  PROC Part96()
    MoveL Offs(pOrigin,43.0,16.5,15.0),vTravel,z5,tPen\WObj:=wPaper;
    MoveL Offs(pOrigin,43.0,16.5,0.0),vApproach,fine,tPen\WObj:=wPaper;
    MoveL Offs(pOrigin,42.8,16.3,0.0),vDraw,z1,tPen\WObj:=wPaper;
    MoveL Offs(pOrigin,42.6,16.5,0.0),vDraw,z1,tPen\WObj:=wPaper;
    MoveL Offs(pOrigin,42.6,18.2,0.0),vDraw,z1,tPen\WObj:=wPaper;
    MoveL Offs(pOrigin,42.8,18.4,0.0),vDraw,z1,tPen\WObj:=wPaper;
    MoveL Offs(pOrigin,43.0,18.2,0.0),vDraw,z1,tPen\WObj:=wPaper;
    MoveL Offs(pOrigin,43.0,17.7,0.0),vDraw,z1,tPen\WObj:=wPaper;
    MoveL Offs(pOrigin,43.2,17.5,0.0),vDraw,z1,tPen\WObj:=wPaper;
    MoveL Offs(pOrigin,43.0,17.3,0.0),vDraw,z1,tPen\WObj:=wPaper;
    MoveL Offs(pOrigin,43.0,16.5,0.0),vDraw,fine,tPen\WObj:=wPaper;
    MoveL Offs(pOrigin,43.0,16.5,15.0),vApproach,z5,tPen\WObj:=wPaper;
    MoveL Offs(pOrigin,43.2,18.4,15.0),vTravel,z5,tPen\WObj:=wPaper;
    MoveL Offs(pOrigin,43.2,18.4,0.0),vApproach,fine,tPen\WObj:=wPaper;
    MoveL Offs(pOrigin,43.0,18.6,0.0),vDraw,z1,tPen\WObj:=wPaper;
    MoveL Offs(pOrigin,43.8,19.2,0.0),vDraw,z1,tPen\WObj:=wPaper;
    MoveL Offs(pOrigin,44.0,19.2,0.0),vDraw,z1,tPen\WObj:=wPaper;
    MoveL Offs(pOrigin,44.2,19.0,0.0),vDraw,z1,tPen\WObj:=wPaper;
    MoveL Offs(pOrigin,44.2,18.8,0.0),vDraw,z1,tPen\WObj:=wPaper;
    MoveL Offs(pOrigin,44.0,18.6,0.0),vDraw,z1,tPen\WObj:=wPaper;
    MoveL Offs(pOrigin,43.6,18.6,0.0),vDraw,z1,tPen\WObj:=wPaper;
    MoveL Offs(pOrigin,43.4,18.4,0.0),vDraw,z1,tPen\WObj:=wPaper;
    MoveL Offs(pOrigin,43.2,18.4,0.0),vDraw,fine,tPen\WObj:=wPaper;
    MoveL Offs(pOrigin,43.2,18.4,15.0),vApproach,z5,tPen\WObj:=wPaper;
    MoveL Offs(pOrigin,46.0,19.0,15.0),vTravel,z5,tPen\WObj:=wPaper;
    MoveL Offs(pOrigin,46.0,19.0,0.0),vApproach,fine,tPen\WObj:=wPaper;
    MoveL Offs(pOrigin,46.2,19.2,0.0),vDraw,z1,tPen\WObj:=wPaper;
    MoveL Offs(pOrigin,46.8,19.2,0.0),vDraw,z1,tPen\WObj:=wPaper;
    MoveL Offs(pOrigin,47.0,19.4,0.0),vDraw,z1,tPen\WObj:=wPaper;
    MoveL Offs(pOrigin,47.6,19.4,0.0),vDraw,z1,tPen\WObj:=wPaper;
    MoveL Offs(pOrigin,47.7,19.5,0.0),vDraw,z1,tPen\WObj:=wPaper;
    MoveL Offs(pOrigin,47.9,19.4,0.0),vDraw,z1,tPen\WObj:=wPaper;
    MoveL Offs(pOrigin,47.9,19.0,0.0),vDraw,z1,tPen\WObj:=wPaper;
    MoveL Offs(pOrigin,47.7,18.8,0.0),vDraw,z1,tPen\WObj:=wPaper;
    MoveL Offs(pOrigin,46.2,18.8,0.0),vDraw,z1,tPen\WObj:=wPaper;
    MoveL Offs(pOrigin,46.0,19.0,0.0),vDraw,fine,tPen\WObj:=wPaper;
    MoveL Offs(pOrigin,46.0,19.0,15.0),vApproach,z5,tPen\WObj:=wPaper;
    MoveL Offs(pOrigin,48.1,19.5,15.0),vTravel,z5,tPen\WObj:=wPaper;
    MoveL Offs(pOrigin,48.1,19.5,0.0),vApproach,fine,tPen\WObj:=wPaper;
    MoveL Offs(pOrigin,48.3,19.7,0.0),vDraw,z1,tPen\WObj:=wPaper;
    MoveL Offs(pOrigin,48.9,19.7,0.0),vDraw,z1,tPen\WObj:=wPaper;
    MoveL Offs(pOrigin,49.1,19.9,0.0),vDraw,z1,tPen\WObj:=wPaper;
    MoveL Offs(pOrigin,49.3,19.9,0.0),vDraw,z1,tPen\WObj:=wPaper;
    MoveL Offs(pOrigin,49.4,19.7,0.0),vDraw,z1,tPen\WObj:=wPaper;
    MoveL Offs(pOrigin,49.4,19.5,0.0),vDraw,z1,tPen\WObj:=wPaper;
    MoveL Offs(pOrigin,49.3,19.4,0.0),vDraw,z1,tPen\WObj:=wPaper;
    MoveL Offs(pOrigin,48.3,19.4,0.0),vDraw,z1,tPen\WObj:=wPaper;
    MoveL Offs(pOrigin,48.1,19.5,0.0),vDraw,fine,tPen\WObj:=wPaper;
    MoveL Offs(pOrigin,48.1,19.5,15.0),vApproach,z5,tPen\WObj:=wPaper;
    MoveL Offs(pOrigin,46.6,26.3,15.0),vTravel,z5,tPen\WObj:=wPaper;
    MoveL Offs(pOrigin,46.6,26.3,0.0),vApproach,fine,tPen\WObj:=wPaper;
    MoveL Offs(pOrigin,46.4,26.5,0.0),vDraw,z1,tPen\WObj:=wPaper;
    MoveL Offs(pOrigin,46.4,27.1,0.0),vDraw,z1,tPen\WObj:=wPaper;
    MoveL Offs(pOrigin,46.2,27.3,0.0),vDraw,z1,tPen\WObj:=wPaper;
    MoveL Offs(pOrigin,46.2,29.9,0.0),vDraw,z1,tPen\WObj:=wPaper;
    MoveL Offs(pOrigin,45.9,30.5,0.0),vDraw,z1,tPen\WObj:=wPaper;
    MoveL Offs(pOrigin,46.0,30.7,0.0),vDraw,z1,tPen\WObj:=wPaper;
    MoveL Offs(pOrigin,46.6,30.7,0.0),vDraw,z1,tPen\WObj:=wPaper;
    MoveL Offs(pOrigin,46.8,30.5,0.0),vDraw,z1,tPen\WObj:=wPaper;
    MoveL Offs(pOrigin,46.8,30.3,0.0),vDraw,z1,tPen\WObj:=wPaper;
    MoveL Offs(pOrigin,46.6,30.1,0.0),vDraw,z1,tPen\WObj:=wPaper;
    MoveL Offs(pOrigin,46.6,28.6,0.0),vDraw,z1,tPen\WObj:=wPaper;
    MoveL Offs(pOrigin,46.8,28.6,0.0),vDraw,z1,tPen\WObj:=wPaper;
    MoveL Offs(pOrigin,47.0,28.4,0.0),vDraw,z1,tPen\WObj:=wPaper;
    MoveL Offs(pOrigin,47.0,27.9,0.0),vDraw,z1,tPen\WObj:=wPaper;
    MoveL Offs(pOrigin,46.8,27.7,0.0),vDraw,z1,tPen\WObj:=wPaper;
    MoveL Offs(pOrigin,46.8,26.5,0.0),vDraw,z1,tPen\WObj:=wPaper;
    MoveL Offs(pOrigin,46.6,26.3,0.0),vDraw,fine,tPen\WObj:=wPaper;
    MoveL Offs(pOrigin,46.6,26.3,15.0),vApproach,z5,tPen\WObj:=wPaper;
    MoveL Offs(pOrigin,47.2,29.0,15.0),vTravel,z5,tPen\WObj:=wPaper;
    MoveL Offs(pOrigin,47.2,29.0,0.0),vApproach,fine,tPen\WObj:=wPaper;
    MoveL Offs(pOrigin,47.0,29.2,0.0),vDraw,z1,tPen\WObj:=wPaper;
    MoveL Offs(pOrigin,47.0,29.7,0.0),vDraw,z1,tPen\WObj:=wPaper;
    MoveL Offs(pOrigin,47.4,30.3,0.0),vDraw,z1,tPen\WObj:=wPaper;
    MoveL Offs(pOrigin,47.6,30.1,0.0),vDraw,z1,tPen\WObj:=wPaper;
    MoveL Offs(pOrigin,47.6,29.7,0.0),vDraw,z1,tPen\WObj:=wPaper;
    MoveL Offs(pOrigin,47.4,29.6,0.0),vDraw,z1,tPen\WObj:=wPaper;
    MoveL Offs(pOrigin,47.4,29.2,0.0),vDraw,z1,tPen\WObj:=wPaper;
    MoveL Offs(pOrigin,47.2,29.0,0.0),vDraw,fine,tPen\WObj:=wPaper;
    MoveL Offs(pOrigin,47.2,29.0,15.0),vApproach,z5,tPen\WObj:=wPaper;
    MoveL Offs(pOrigin,46.4,31.6,15.0),vTravel,z5,tPen\WObj:=wPaper;
    MoveL Offs(pOrigin,46.4,31.6,0.0),vApproach,fine,tPen\WObj:=wPaper;
    MoveL Offs(pOrigin,46.2,31.8,0.0),vDraw,z1,tPen\WObj:=wPaper;
    MoveL Offs(pOrigin,46.2,32.2,0.0),vDraw,z1,tPen\WObj:=wPaper;
    MoveL Offs(pOrigin,46.0,32.4,0.0),vDraw,z1,tPen\WObj:=wPaper;
    MoveL Offs(pOrigin,46.0,33.0,0.0),vDraw,z1,tPen\WObj:=wPaper;
    MoveL Offs(pOrigin,45.9,33.1,0.0),vDraw,z1,tPen\WObj:=wPaper;
    MoveL Offs(pOrigin,45.9,33.9,0.0),vDraw,z1,tPen\WObj:=wPaper;
    MoveL Offs(pOrigin,45.7,34.1,0.0),vDraw,z1,tPen\WObj:=wPaper;
    MoveL Offs(pOrigin,45.7,35.0,0.0),vDraw,z1,tPen\WObj:=wPaper;
    MoveL Offs(pOrigin,45.5,35.2,0.0),vDraw,z1,tPen\WObj:=wPaper;
    MoveL Offs(pOrigin,45.5,37.3,0.0),vDraw,z1,tPen\WObj:=wPaper;
    MoveL Offs(pOrigin,45.7,37.5,0.0),vDraw,z1,tPen\WObj:=wPaper;
    MoveL Offs(pOrigin,45.7,38.1,0.0),vDraw,z1,tPen\WObj:=wPaper;
    MoveL Offs(pOrigin,45.9,38.2,0.0),vDraw,z1,tPen\WObj:=wPaper;
    MoveL Offs(pOrigin,45.9,38.8,0.0),vDraw,z1,tPen\WObj:=wPaper;
    MoveL Offs(pOrigin,46.0,39.0,0.0),vDraw,z1,tPen\WObj:=wPaper;
    MoveL Offs(pOrigin,46.0,39.2,0.0),vDraw,z1,tPen\WObj:=wPaper;
    MoveL Offs(pOrigin,46.2,39.4,0.0),vDraw,z1,tPen\WObj:=wPaper;
    MoveL Offs(pOrigin,46.8,40.7,0.0),vDraw,z1,tPen\WObj:=wPaper;
    MoveL Offs(pOrigin,47.4,41.5,0.0),vDraw,z1,tPen\WObj:=wPaper;
    MoveL Offs(pOrigin,47.6,41.3,0.0),vDraw,z1,tPen\WObj:=wPaper;
    MoveL Offs(pOrigin,47.6,40.7,0.0),vDraw,z1,tPen\WObj:=wPaper;
    MoveL Offs(pOrigin,48.3,40.7,0.0),vDraw,z1,tPen\WObj:=wPaper;
    MoveL Offs(pOrigin,48.5,40.5,0.0),vDraw,z1,tPen\WObj:=wPaper;
    MoveL Offs(pOrigin,47.6,39.6,0.0),vDraw,z1,tPen\WObj:=wPaper;
    MoveL Offs(pOrigin,47.6,39.4,0.0),vDraw,z1,tPen\WObj:=wPaper;
    MoveL Offs(pOrigin,46.6,38.2,0.0),vDraw,z1,tPen\WObj:=wPaper;
    MoveL Offs(pOrigin,46.6,38.1,0.0),vDraw,z1,tPen\WObj:=wPaper;
    MoveL Offs(pOrigin,46.4,37.9,0.0),vDraw,z1,tPen\WObj:=wPaper;
    MoveL Offs(pOrigin,46.4,37.5,0.0),vDraw,z1,tPen\WObj:=wPaper;
    MoveL Offs(pOrigin,45.9,36.5,0.0),vDraw,z1,tPen\WObj:=wPaper;
    MoveL Offs(pOrigin,45.9,35.4,0.0),vDraw,z1,tPen\WObj:=wPaper;
    MoveL Offs(pOrigin,46.6,35.4,0.0),vDraw,z1,tPen\WObj:=wPaper;
    MoveL Offs(pOrigin,46.6,35.6,0.0),vDraw,z1,tPen\WObj:=wPaper;
    MoveL Offs(pOrigin,46.8,35.8,0.0),vDraw,z1,tPen\WObj:=wPaper;
    MoveL Offs(pOrigin,47.4,37.1,0.0),vDraw,z1,tPen\WObj:=wPaper;
    MoveL Offs(pOrigin,47.7,37.5,0.0),vDraw,z1,tPen\WObj:=wPaper;
    MoveL Offs(pOrigin,47.7,37.7,0.0),vDraw,z1,tPen\WObj:=wPaper;
    MoveL Offs(pOrigin,48.1,38.1,0.0),vDraw,z1,tPen\WObj:=wPaper;
  ENDPROC

  PROC Part97()
    MoveL Offs(pOrigin,48.1,38.2,0.0),vDraw,z1,tPen\WObj:=wPaper;
    MoveL Offs(pOrigin,51.1,41.3,0.0),vDraw,z1,tPen\WObj:=wPaper;
    MoveL Offs(pOrigin,51.3,41.3,0.0),vDraw,z1,tPen\WObj:=wPaper;
    MoveL Offs(pOrigin,52.3,42.2,0.0),vDraw,z1,tPen\WObj:=wPaper;
    MoveL Offs(pOrigin,52.5,42.2,0.0),vDraw,z1,tPen\WObj:=wPaper;
    MoveL Offs(pOrigin,53.0,42.8,0.0),vDraw,z1,tPen\WObj:=wPaper;
    MoveL Offs(pOrigin,53.2,42.8,0.0),vDraw,z1,tPen\WObj:=wPaper;
    MoveL Offs(pOrigin,53.4,42.6,0.0),vDraw,z1,tPen\WObj:=wPaper;
    MoveL Offs(pOrigin,52.5,41.5,0.0),vDraw,z1,tPen\WObj:=wPaper;
    MoveL Offs(pOrigin,52.5,41.3,0.0),vDraw,z1,tPen\WObj:=wPaper;
    MoveL Offs(pOrigin,51.7,40.3,0.0),vDraw,z1,tPen\WObj:=wPaper;
    MoveL Offs(pOrigin,51.5,39.8,0.0),vDraw,z1,tPen\WObj:=wPaper;
    MoveL Offs(pOrigin,51.1,39.4,0.0),vDraw,z1,tPen\WObj:=wPaper;
    MoveL Offs(pOrigin,51.1,39.2,0.0),vDraw,z1,tPen\WObj:=wPaper;
    MoveL Offs(pOrigin,50.2,37.5,0.0),vDraw,z1,tPen\WObj:=wPaper;
    MoveL Offs(pOrigin,50.2,37.1,0.0),vDraw,z1,tPen\WObj:=wPaper;
    MoveL Offs(pOrigin,49.8,36.7,0.0),vDraw,z1,tPen\WObj:=wPaper;
    MoveL Offs(pOrigin,49.6,36.7,0.0),vDraw,z1,tPen\WObj:=wPaper;
    MoveL Offs(pOrigin,49.4,36.9,0.0),vDraw,z1,tPen\WObj:=wPaper;
    MoveL Offs(pOrigin,49.1,36.9,0.0),vDraw,z1,tPen\WObj:=wPaper;
    MoveL Offs(pOrigin,49.1,36.7,0.0),vDraw,z1,tPen\WObj:=wPaper;
    MoveL Offs(pOrigin,48.5,36.0,0.0),vDraw,z1,tPen\WObj:=wPaper;
    MoveL Offs(pOrigin,48.5,35.8,0.0),vDraw,z1,tPen\WObj:=wPaper;
    MoveL Offs(pOrigin,48.3,35.6,0.0),vDraw,z1,tPen\WObj:=wPaper;
    MoveL Offs(pOrigin,48.3,35.4,0.0),vDraw,z1,tPen\WObj:=wPaper;
    MoveL Offs(pOrigin,48.1,35.2,0.0),vDraw,z1,tPen\WObj:=wPaper;
    MoveL Offs(pOrigin,48.1,35.0,0.0),vDraw,z1,tPen\WObj:=wPaper;
    MoveL Offs(pOrigin,47.9,34.8,0.0),vDraw,z1,tPen\WObj:=wPaper;
    MoveL Offs(pOrigin,47.9,34.7,0.0),vDraw,z1,tPen\WObj:=wPaper;
    MoveL Offs(pOrigin,46.8,32.6,0.0),vDraw,z1,tPen\WObj:=wPaper;
    MoveL Offs(pOrigin,46.8,32.2,0.0),vDraw,z1,tPen\WObj:=wPaper;
    MoveL Offs(pOrigin,46.4,31.6,0.0),vDraw,fine,tPen\WObj:=wPaper;
    MoveL Offs(pOrigin,46.4,31.6,15.0),vApproach,z5,tPen\WObj:=wPaper;
    MoveL Offs(pOrigin,45.1,33.5,15.0),vTravel,z5,tPen\WObj:=wPaper;
    MoveL Offs(pOrigin,45.1,33.5,0.0),vApproach,fine,tPen\WObj:=wPaper;
    MoveL Offs(pOrigin,44.9,33.7,0.0),vDraw,z1,tPen\WObj:=wPaper;
    MoveL Offs(pOrigin,44.9,34.7,0.0),vDraw,z1,tPen\WObj:=wPaper;
    MoveL Offs(pOrigin,45.1,34.8,0.0),vDraw,z1,tPen\WObj:=wPaper;
    MoveL Offs(pOrigin,45.3,34.7,0.0),vDraw,z1,tPen\WObj:=wPaper;
    MoveL Offs(pOrigin,45.3,33.7,0.0),vDraw,z1,tPen\WObj:=wPaper;
    MoveL Offs(pOrigin,45.1,33.5,0.0),vDraw,fine,tPen\WObj:=wPaper;
    MoveL Offs(pOrigin,45.1,33.5,15.0),vApproach,z5,tPen\WObj:=wPaper;
    MoveL Offs(pOrigin,44.9,34.7,15.0),vTravel,z5,tPen\WObj:=wPaper;
    MoveL Offs(pOrigin,44.9,34.7,0.0),vApproach,fine,tPen\WObj:=wPaper;
    MoveL Offs(pOrigin,44.7,34.8,0.0),vDraw,z1,tPen\WObj:=wPaper;
    MoveL Offs(pOrigin,44.7,37.5,0.0),vDraw,z1,tPen\WObj:=wPaper;
    MoveL Offs(pOrigin,44.9,37.7,0.0),vDraw,z1,tPen\WObj:=wPaper;
    MoveL Offs(pOrigin,45.1,37.5,0.0),vDraw,z1,tPen\WObj:=wPaper;
    MoveL Offs(pOrigin,45.1,34.8,0.0),vDraw,z1,tPen\WObj:=wPaper;
    MoveL Offs(pOrigin,44.9,34.7,0.0),vDraw,fine,tPen\WObj:=wPaper;
    MoveL Offs(pOrigin,44.9,34.7,15.0),vApproach,z5,tPen\WObj:=wPaper;
    MoveL Offs(pOrigin,57.4,15.6,15.0),vTravel,z5,tPen\WObj:=wPaper;
    MoveL Offs(pOrigin,57.4,15.6,0.0),vApproach,fine,tPen\WObj:=wPaper;
    MoveL Offs(pOrigin,58.3,15.6,0.0),vDraw,z1,tPen\WObj:=wPaper;
    MoveL Offs(pOrigin,58.5,15.4,0.0),vDraw,z1,tPen\WObj:=wPaper;
    MoveL Offs(pOrigin,58.3,15.2,0.0),vDraw,z1,tPen\WObj:=wPaper;
    MoveL Offs(pOrigin,57.4,15.2,0.0),vDraw,z1,tPen\WObj:=wPaper;
    MoveL Offs(pOrigin,57.2,15.4,0.0),vDraw,z1,tPen\WObj:=wPaper;
    MoveL Offs(pOrigin,57.4,15.6,0.0),vDraw,fine,tPen\WObj:=wPaper;
    MoveL Offs(pOrigin,57.4,15.6,15.0),vApproach,z5,tPen\WObj:=wPaper;
    MoveL Offs(pOrigin,57.4,14.8,15.0),vTravel,z5,tPen\WObj:=wPaper;
    MoveL Offs(pOrigin,57.4,14.8,0.0),vApproach,fine,tPen\WObj:=wPaper;
    MoveL Offs(pOrigin,58.7,14.8,0.0),vDraw,z1,tPen\WObj:=wPaper;
    MoveL Offs(pOrigin,58.9,14.6,0.0),vDraw,z1,tPen\WObj:=wPaper;
    MoveL Offs(pOrigin,58.7,14.4,0.0),vDraw,z1,tPen\WObj:=wPaper;
    MoveL Offs(pOrigin,57.4,14.4,0.0),vDraw,z1,tPen\WObj:=wPaper;
    MoveL Offs(pOrigin,57.2,14.6,0.0),vDraw,z1,tPen\WObj:=wPaper;
    MoveL Offs(pOrigin,57.4,14.8,0.0),vDraw,fine,tPen\WObj:=wPaper;
    MoveL Offs(pOrigin,57.4,14.8,15.0),vApproach,z5,tPen\WObj:=wPaper;
    MoveL Offs(pOrigin,59.1,14.4,15.0),vTravel,z5,tPen\WObj:=wPaper;
    MoveL Offs(pOrigin,59.1,14.4,0.0),vApproach,fine,tPen\WObj:=wPaper;
    MoveL Offs(pOrigin,59.3,14.6,0.0),vDraw,z1,tPen\WObj:=wPaper;
    MoveL Offs(pOrigin,60.6,14.6,0.0),vDraw,z1,tPen\WObj:=wPaper;
    MoveL Offs(pOrigin,60.8,14.4,0.0),vDraw,z1,tPen\WObj:=wPaper;
    MoveL Offs(pOrigin,60.6,14.3,0.0),vDraw,z1,tPen\WObj:=wPaper;
    MoveL Offs(pOrigin,59.3,14.3,0.0),vDraw,z1,tPen\WObj:=wPaper;
    MoveL Offs(pOrigin,59.1,14.4,0.0),vDraw,fine,tPen\WObj:=wPaper;
    MoveL Offs(pOrigin,59.1,14.4,15.0),vApproach,z5,tPen\WObj:=wPaper;
    MoveL Offs(pOrigin,59.3,15.0,15.0),vTravel,z5,tPen\WObj:=wPaper;
    MoveL Offs(pOrigin,59.3,15.0,0.0),vApproach,fine,tPen\WObj:=wPaper;
    MoveL Offs(pOrigin,59.1,15.2,0.0),vDraw,z1,tPen\WObj:=wPaper;
    MoveL Offs(pOrigin,59.3,15.4,0.0),vDraw,z1,tPen\WObj:=wPaper;
    MoveL Offs(pOrigin,60.2,15.4,0.0),vDraw,z1,tPen\WObj:=wPaper;
    MoveL Offs(pOrigin,60.4,15.2,0.0),vDraw,z1,tPen\WObj:=wPaper;
    MoveL Offs(pOrigin,60.2,15.0,0.0),vDraw,z1,tPen\WObj:=wPaper;
    MoveL Offs(pOrigin,59.3,15.0,0.0),vDraw,fine,tPen\WObj:=wPaper;
    MoveL Offs(pOrigin,59.3,15.0,15.0),vApproach,z5,tPen\WObj:=wPaper;
    MoveL Offs(pOrigin,61.0,15.0,15.0),vTravel,z5,tPen\WObj:=wPaper;
    MoveL Offs(pOrigin,61.0,15.0,0.0),vApproach,fine,tPen\WObj:=wPaper;
    MoveL Offs(pOrigin,61.2,15.2,0.0),vDraw,z1,tPen\WObj:=wPaper;
    MoveL Offs(pOrigin,61.9,15.2,0.0),vDraw,z1,tPen\WObj:=wPaper;
    MoveL Offs(pOrigin,62.1,15.0,0.0),vDraw,z1,tPen\WObj:=wPaper;
    MoveL Offs(pOrigin,61.9,14.8,0.0),vDraw,z1,tPen\WObj:=wPaper;
    MoveL Offs(pOrigin,61.2,14.8,0.0),vDraw,z1,tPen\WObj:=wPaper;
    MoveL Offs(pOrigin,61.0,15.0,0.0),vDraw,fine,tPen\WObj:=wPaper;
    MoveL Offs(pOrigin,61.0,15.0,15.0),vApproach,z5,tPen\WObj:=wPaper;
    MoveL Offs(pOrigin,61.2,14.4,15.0),vTravel,z5,tPen\WObj:=wPaper;
    MoveL Offs(pOrigin,61.2,14.4,0.0),vApproach,fine,tPen\WObj:=wPaper;
    MoveL Offs(pOrigin,62.5,14.4,0.0),vDraw,z1,tPen\WObj:=wPaper;
    MoveL Offs(pOrigin,62.7,14.3,0.0),vDraw,z1,tPen\WObj:=wPaper;
    MoveL Offs(pOrigin,62.5,14.1,0.0),vDraw,z1,tPen\WObj:=wPaper;
    MoveL Offs(pOrigin,61.2,14.1,0.0),vDraw,z1,tPen\WObj:=wPaper;
    MoveL Offs(pOrigin,61.0,14.3,0.0),vDraw,z1,tPen\WObj:=wPaper;
    MoveL Offs(pOrigin,61.2,14.4,0.0),vDraw,fine,tPen\WObj:=wPaper;
    MoveL Offs(pOrigin,61.2,14.4,15.0),vApproach,z5,tPen\WObj:=wPaper;
    MoveL Offs(pOrigin,62.9,14.1,15.0),vTravel,z5,tPen\WObj:=wPaper;
    MoveL Offs(pOrigin,62.9,14.1,0.0),vApproach,fine,tPen\WObj:=wPaper;
    MoveL Offs(pOrigin,63.0,14.3,0.0),vDraw,z1,tPen\WObj:=wPaper;
    MoveL Offs(pOrigin,64.4,14.3,0.0),vDraw,z1,tPen\WObj:=wPaper;
    MoveL Offs(pOrigin,64.6,14.1,0.0),vDraw,z1,tPen\WObj:=wPaper;
    MoveL Offs(pOrigin,64.4,13.9,0.0),vDraw,z1,tPen\WObj:=wPaper;
    MoveL Offs(pOrigin,63.0,13.9,0.0),vDraw,z1,tPen\WObj:=wPaper;
    MoveL Offs(pOrigin,62.9,14.1,0.0),vDraw,fine,tPen\WObj:=wPaper;
    MoveL Offs(pOrigin,62.9,14.1,15.0),vApproach,z5,tPen\WObj:=wPaper;
    MoveL Offs(pOrigin,63.0,14.6,15.0),vTravel,z5,tPen\WObj:=wPaper;
    MoveL Offs(pOrigin,63.0,14.6,0.0),vApproach,fine,tPen\WObj:=wPaper;
    MoveL Offs(pOrigin,62.9,14.8,0.0),vDraw,z1,tPen\WObj:=wPaper;
    MoveL Offs(pOrigin,63.0,15.0,0.0),vDraw,z1,tPen\WObj:=wPaper;
    MoveL Offs(pOrigin,63.8,15.0,0.0),vDraw,z1,tPen\WObj:=wPaper;
    MoveL Offs(pOrigin,64.0,14.8,0.0),vDraw,z1,tPen\WObj:=wPaper;
  ENDPROC

  PROC Part98()
    MoveL Offs(pOrigin,63.8,14.6,0.0),vDraw,z1,tPen\WObj:=wPaper;
    MoveL Offs(pOrigin,63.0,14.6,0.0),vDraw,fine,tPen\WObj:=wPaper;
    MoveL Offs(pOrigin,63.0,14.6,15.0),vApproach,z5,tPen\WObj:=wPaper;
    MoveL Offs(pOrigin,64.7,14.6,15.0),vTravel,z5,tPen\WObj:=wPaper;
    MoveL Offs(pOrigin,64.7,14.6,0.0),vApproach,fine,tPen\WObj:=wPaper;
    MoveL Offs(pOrigin,64.9,14.8,0.0),vDraw,z1,tPen\WObj:=wPaper;
    MoveL Offs(pOrigin,65.7,14.8,0.0),vDraw,z1,tPen\WObj:=wPaper;
    MoveL Offs(pOrigin,65.9,14.6,0.0),vDraw,z1,tPen\WObj:=wPaper;
    MoveL Offs(pOrigin,65.7,14.4,0.0),vDraw,z1,tPen\WObj:=wPaper;
    MoveL Offs(pOrigin,64.9,14.4,0.0),vDraw,z1,tPen\WObj:=wPaper;
    MoveL Offs(pOrigin,64.7,14.6,0.0),vDraw,fine,tPen\WObj:=wPaper;
    MoveL Offs(pOrigin,64.7,14.6,15.0),vApproach,z5,tPen\WObj:=wPaper;
    MoveL Offs(pOrigin,64.9,14.1,15.0),vTravel,z5,tPen\WObj:=wPaper;
    MoveL Offs(pOrigin,64.9,14.1,0.0),vApproach,fine,tPen\WObj:=wPaper;
    MoveL Offs(pOrigin,66.1,14.1,0.0),vDraw,z1,tPen\WObj:=wPaper;
    MoveL Offs(pOrigin,66.3,13.9,0.0),vDraw,z1,tPen\WObj:=wPaper;
    MoveL Offs(pOrigin,66.1,13.7,0.0),vDraw,z1,tPen\WObj:=wPaper;
    MoveL Offs(pOrigin,64.9,13.7,0.0),vDraw,z1,tPen\WObj:=wPaper;
    MoveL Offs(pOrigin,64.7,13.9,0.0),vDraw,z1,tPen\WObj:=wPaper;
    MoveL Offs(pOrigin,64.9,14.1,0.0),vDraw,fine,tPen\WObj:=wPaper;
    MoveL Offs(pOrigin,64.9,14.1,15.0),vApproach,z5,tPen\WObj:=wPaper;
    MoveL Offs(pOrigin,66.4,13.7,15.0),vTravel,z5,tPen\WObj:=wPaper;
    MoveL Offs(pOrigin,66.4,13.7,0.0),vApproach,fine,tPen\WObj:=wPaper;
    MoveL Offs(pOrigin,66.6,13.9,0.0),vDraw,z1,tPen\WObj:=wPaper;
    MoveL Offs(pOrigin,68.0,13.9,0.0),vDraw,z1,tPen\WObj:=wPaper;
    MoveL Offs(pOrigin,68.1,13.7,0.0),vDraw,z1,tPen\WObj:=wPaper;
    MoveL Offs(pOrigin,68.0,13.5,0.0),vDraw,z1,tPen\WObj:=wPaper;
    MoveL Offs(pOrigin,66.6,13.5,0.0),vDraw,z1,tPen\WObj:=wPaper;
    MoveL Offs(pOrigin,66.4,13.7,0.0),vDraw,fine,tPen\WObj:=wPaper;
    MoveL Offs(pOrigin,66.4,13.7,15.0),vApproach,z5,tPen\WObj:=wPaper;
    MoveL Offs(pOrigin,66.6,14.3,15.0),vTravel,z5,tPen\WObj:=wPaper;
    MoveL Offs(pOrigin,66.6,14.3,0.0),vApproach,fine,tPen\WObj:=wPaper;
    MoveL Offs(pOrigin,66.4,14.4,0.0),vDraw,z1,tPen\WObj:=wPaper;
    MoveL Offs(pOrigin,66.6,14.6,0.0),vDraw,z1,tPen\WObj:=wPaper;
    MoveL Offs(pOrigin,67.6,14.6,0.0),vDraw,z1,tPen\WObj:=wPaper;
    MoveL Offs(pOrigin,67.8,14.4,0.0),vDraw,z1,tPen\WObj:=wPaper;
    MoveL Offs(pOrigin,67.6,14.3,0.0),vDraw,z1,tPen\WObj:=wPaper;
    MoveL Offs(pOrigin,66.6,14.3,0.0),vDraw,fine,tPen\WObj:=wPaper;
    MoveL Offs(pOrigin,66.6,14.3,15.0),vApproach,z5,tPen\WObj:=wPaper;
    MoveL Offs(pOrigin,66.4,15.6,15.0),vTravel,z5,tPen\WObj:=wPaper;
    MoveL Offs(pOrigin,66.4,15.6,0.0),vApproach,fine,tPen\WObj:=wPaper;
    MoveL Offs(pOrigin,66.3,15.8,0.0),vDraw,z1,tPen\WObj:=wPaper;
    MoveL Offs(pOrigin,66.4,16.0,0.0),vDraw,z1,tPen\WObj:=wPaper;
    MoveL Offs(pOrigin,67.2,16.0,0.0),vDraw,z1,tPen\WObj:=wPaper;
    MoveL Offs(pOrigin,67.4,15.8,0.0),vDraw,z1,tPen\WObj:=wPaper;
    MoveL Offs(pOrigin,67.2,15.6,0.0),vDraw,z1,tPen\WObj:=wPaper;
    MoveL Offs(pOrigin,66.4,15.6,0.0),vDraw,fine,tPen\WObj:=wPaper;
    MoveL Offs(pOrigin,66.4,15.6,15.0),vApproach,z5,tPen\WObj:=wPaper;
    MoveL Offs(pOrigin,65.5,16.0,15.0),vTravel,z5,tPen\WObj:=wPaper;
    MoveL Offs(pOrigin,65.5,16.0,0.0),vApproach,fine,tPen\WObj:=wPaper;
    MoveL Offs(pOrigin,65.3,15.8,0.0),vDraw,z1,tPen\WObj:=wPaper;
    MoveL Offs(pOrigin,64.6,15.8,0.0),vDraw,z1,tPen\WObj:=wPaper;
    MoveL Offs(pOrigin,64.4,16.0,0.0),vDraw,z1,tPen\WObj:=wPaper;
    MoveL Offs(pOrigin,64.6,16.1,0.0),vDraw,z1,tPen\WObj:=wPaper;
    MoveL Offs(pOrigin,65.3,16.1,0.0),vDraw,z1,tPen\WObj:=wPaper;
    MoveL Offs(pOrigin,65.5,16.0,0.0),vDraw,fine,tPen\WObj:=wPaper;
    MoveL Offs(pOrigin,65.5,16.0,15.0),vApproach,z5,tPen\WObj:=wPaper;
    MoveL Offs(pOrigin,68.1,15.6,15.0),vTravel,z5,tPen\WObj:=wPaper;
    MoveL Offs(pOrigin,68.1,15.6,0.0),vApproach,fine,tPen\WObj:=wPaper;
    MoveL Offs(pOrigin,68.3,15.8,0.0),vDraw,z1,tPen\WObj:=wPaper;
    MoveL Offs(pOrigin,69.1,15.8,0.0),vDraw,z1,tPen\WObj:=wPaper;
    MoveL Offs(pOrigin,69.3,15.6,0.0),vDraw,z1,tPen\WObj:=wPaper;
    MoveL Offs(pOrigin,69.1,15.4,0.0),vDraw,z1,tPen\WObj:=wPaper;
    MoveL Offs(pOrigin,68.3,15.4,0.0),vDraw,z1,tPen\WObj:=wPaper;
    MoveL Offs(pOrigin,68.1,15.6,0.0),vDraw,fine,tPen\WObj:=wPaper;
    MoveL Offs(pOrigin,68.1,15.6,15.0),vApproach,z5,tPen\WObj:=wPaper;
    MoveL Offs(pOrigin,68.5,14.4,15.0),vTravel,z5,tPen\WObj:=wPaper;
    MoveL Offs(pOrigin,68.5,14.4,0.0),vApproach,fine,tPen\WObj:=wPaper;
    MoveL Offs(pOrigin,69.3,14.4,0.0),vDraw,z1,tPen\WObj:=wPaper;
    MoveL Offs(pOrigin,69.5,14.3,0.0),vDraw,z1,tPen\WObj:=wPaper;
    MoveL Offs(pOrigin,69.3,14.1,0.0),vDraw,z1,tPen\WObj:=wPaper;
    MoveL Offs(pOrigin,68.5,14.1,0.0),vDraw,z1,tPen\WObj:=wPaper;
    MoveL Offs(pOrigin,68.3,14.3,0.0),vDraw,z1,tPen\WObj:=wPaper;
    MoveL Offs(pOrigin,68.5,14.4,0.0),vDraw,fine,tPen\WObj:=wPaper;
    MoveL Offs(pOrigin,68.5,14.4,15.0),vApproach,z5,tPen\WObj:=wPaper;
    MoveL Offs(pOrigin,68.3,13.7,15.0),vTravel,z5,tPen\WObj:=wPaper;
    MoveL Offs(pOrigin,68.3,13.7,0.0),vApproach,fine,tPen\WObj:=wPaper;
    MoveL Offs(pOrigin,69.7,13.7,0.0),vDraw,z1,tPen\WObj:=wPaper;
    MoveL Offs(pOrigin,69.8,13.5,0.0),vDraw,z1,tPen\WObj:=wPaper;
    MoveL Offs(pOrigin,69.7,13.3,0.0),vDraw,z1,tPen\WObj:=wPaper;
    MoveL Offs(pOrigin,68.3,13.3,0.0),vDraw,z1,tPen\WObj:=wPaper;
    MoveL Offs(pOrigin,68.1,13.5,0.0),vDraw,z1,tPen\WObj:=wPaper;
    MoveL Offs(pOrigin,68.3,13.7,0.0),vDraw,fine,tPen\WObj:=wPaper;
    MoveL Offs(pOrigin,68.3,13.7,15.0),vApproach,z5,tPen\WObj:=wPaper;
    MoveL Offs(pOrigin,70.0,13.3,15.0),vTravel,z5,tPen\WObj:=wPaper;
    MoveL Offs(pOrigin,70.0,13.3,0.0),vApproach,fine,tPen\WObj:=wPaper;
    MoveL Offs(pOrigin,70.2,13.5,0.0),vDraw,z1,tPen\WObj:=wPaper;
    MoveL Offs(pOrigin,71.5,13.5,0.0),vDraw,z1,tPen\WObj:=wPaper;
    MoveL Offs(pOrigin,71.7,13.3,0.0),vDraw,z1,tPen\WObj:=wPaper;
    MoveL Offs(pOrigin,71.5,13.1,0.0),vDraw,z1,tPen\WObj:=wPaper;
    MoveL Offs(pOrigin,70.2,13.1,0.0),vDraw,z1,tPen\WObj:=wPaper;
    MoveL Offs(pOrigin,70.0,13.3,0.0),vDraw,fine,tPen\WObj:=wPaper;
    MoveL Offs(pOrigin,70.0,13.3,15.0),vApproach,z5,tPen\WObj:=wPaper;
    MoveL Offs(pOrigin,70.2,13.9,15.0),vTravel,z5,tPen\WObj:=wPaper;
    MoveL Offs(pOrigin,70.2,13.9,0.0),vApproach,fine,tPen\WObj:=wPaper;
    MoveL Offs(pOrigin,70.0,14.1,0.0),vDraw,z1,tPen\WObj:=wPaper;
    MoveL Offs(pOrigin,70.2,14.3,0.0),vDraw,z1,tPen\WObj:=wPaper;
    MoveL Offs(pOrigin,71.2,14.3,0.0),vDraw,z1,tPen\WObj:=wPaper;
    MoveL Offs(pOrigin,71.4,14.1,0.0),vDraw,z1,tPen\WObj:=wPaper;
    MoveL Offs(pOrigin,71.2,13.9,0.0),vDraw,z1,tPen\WObj:=wPaper;
    MoveL Offs(pOrigin,70.2,13.9,0.0),vDraw,fine,tPen\WObj:=wPaper;
    MoveL Offs(pOrigin,70.2,13.9,15.0),vApproach,z5,tPen\WObj:=wPaper;
    MoveL Offs(pOrigin,70.2,15.2,15.0),vTravel,z5,tPen\WObj:=wPaper;
    MoveL Offs(pOrigin,70.2,15.2,0.0),vApproach,fine,tPen\WObj:=wPaper;
    MoveL Offs(pOrigin,70.0,15.4,0.0),vDraw,z1,tPen\WObj:=wPaper;
    MoveL Offs(pOrigin,70.2,15.6,0.0),vDraw,z1,tPen\WObj:=wPaper;
    MoveL Offs(pOrigin,71.2,15.6,0.0),vDraw,z1,tPen\WObj:=wPaper;
    MoveL Offs(pOrigin,71.4,15.4,0.0),vDraw,z1,tPen\WObj:=wPaper;
    MoveL Offs(pOrigin,71.2,15.2,0.0),vDraw,z1,tPen\WObj:=wPaper;
    MoveL Offs(pOrigin,70.2,15.2,0.0),vDraw,fine,tPen\WObj:=wPaper;
    MoveL Offs(pOrigin,70.2,15.2,15.0),vApproach,z5,tPen\WObj:=wPaper;
    MoveL Offs(pOrigin,71.9,15.2,15.0),vTravel,z5,tPen\WObj:=wPaper;
    MoveL Offs(pOrigin,71.9,15.2,0.0),vApproach,fine,tPen\WObj:=wPaper;
    MoveL Offs(pOrigin,72.1,15.4,0.0),vDraw,z1,tPen\WObj:=wPaper;
    MoveL Offs(pOrigin,73.1,15.4,0.0),vDraw,z1,tPen\WObj:=wPaper;
    MoveL Offs(pOrigin,73.2,15.2,0.0),vDraw,z1,tPen\WObj:=wPaper;
    MoveL Offs(pOrigin,73.1,15.0,0.0),vDraw,z1,tPen\WObj:=wPaper;
    MoveL Offs(pOrigin,72.1,15.0,0.0),vDraw,z1,tPen\WObj:=wPaper;
    MoveL Offs(pOrigin,71.9,15.2,0.0),vDraw,fine,tPen\WObj:=wPaper;
    MoveL Offs(pOrigin,71.9,15.2,15.0),vApproach,z5,tPen\WObj:=wPaper;
  ENDPROC

  PROC Part99()
    MoveL Offs(pOrigin,72.1,14.1,15.0),vTravel,z5,tPen\WObj:=wPaper;
    MoveL Offs(pOrigin,72.1,14.1,0.0),vApproach,fine,tPen\WObj:=wPaper;
    MoveL Offs(pOrigin,73.1,14.1,0.0),vDraw,z1,tPen\WObj:=wPaper;
    MoveL Offs(pOrigin,73.2,13.9,0.0),vDraw,z1,tPen\WObj:=wPaper;
    MoveL Offs(pOrigin,73.1,13.7,0.0),vDraw,z1,tPen\WObj:=wPaper;
    MoveL Offs(pOrigin,72.1,13.7,0.0),vDraw,z1,tPen\WObj:=wPaper;
    MoveL Offs(pOrigin,71.9,13.9,0.0),vDraw,z1,tPen\WObj:=wPaper;
    MoveL Offs(pOrigin,72.1,14.1,0.0),vDraw,fine,tPen\WObj:=wPaper;
    MoveL Offs(pOrigin,72.1,14.1,15.0),vApproach,z5,tPen\WObj:=wPaper;
    MoveL Offs(pOrigin,72.1,13.3,15.0),vTravel,z5,tPen\WObj:=wPaper;
    MoveL Offs(pOrigin,72.1,13.3,0.0),vApproach,fine,tPen\WObj:=wPaper;
    MoveL Offs(pOrigin,73.4,13.3,0.0),vDraw,z1,tPen\WObj:=wPaper;
    MoveL Offs(pOrigin,73.6,13.1,0.0),vDraw,z1,tPen\WObj:=wPaper;
    MoveL Offs(pOrigin,73.4,12.9,0.0),vDraw,z1,tPen\WObj:=wPaper;
    MoveL Offs(pOrigin,72.1,12.9,0.0),vDraw,z1,tPen\WObj:=wPaper;
    MoveL Offs(pOrigin,71.9,13.1,0.0),vDraw,z1,tPen\WObj:=wPaper;
    MoveL Offs(pOrigin,72.1,13.3,0.0),vDraw,fine,tPen\WObj:=wPaper;
    MoveL Offs(pOrigin,72.1,13.3,15.0),vApproach,z5,tPen\WObj:=wPaper;
    MoveL Offs(pOrigin,73.8,12.9,15.0),vTravel,z5,tPen\WObj:=wPaper;
    MoveL Offs(pOrigin,73.8,12.9,0.0),vApproach,fine,tPen\WObj:=wPaper;
    MoveL Offs(pOrigin,74.0,13.1,0.0),vDraw,z1,tPen\WObj:=wPaper;
    MoveL Offs(pOrigin,75.3,13.1,0.0),vDraw,z1,tPen\WObj:=wPaper;
    MoveL Offs(pOrigin,75.5,12.9,0.0),vDraw,z1,tPen\WObj:=wPaper;
    MoveL Offs(pOrigin,75.3,12.7,0.0),vDraw,z1,tPen\WObj:=wPaper;
    MoveL Offs(pOrigin,74.0,12.7,0.0),vDraw,z1,tPen\WObj:=wPaper;
    MoveL Offs(pOrigin,73.8,12.9,0.0),vDraw,fine,tPen\WObj:=wPaper;
    MoveL Offs(pOrigin,73.8,12.9,15.0),vApproach,z5,tPen\WObj:=wPaper;
    MoveL Offs(pOrigin,74.0,13.5,15.0),vTravel,z5,tPen\WObj:=wPaper;
    MoveL Offs(pOrigin,74.0,13.5,0.0),vApproach,fine,tPen\WObj:=wPaper;
    MoveL Offs(pOrigin,73.8,13.7,0.0),vDraw,z1,tPen\WObj:=wPaper;
    MoveL Offs(pOrigin,74.0,13.9,0.0),vDraw,z1,tPen\WObj:=wPaper;
    MoveL Offs(pOrigin,74.9,13.9,0.0),vDraw,z1,tPen\WObj:=wPaper;
    MoveL Offs(pOrigin,75.1,13.7,0.0),vDraw,z1,tPen\WObj:=wPaper;
    MoveL Offs(pOrigin,74.9,13.5,0.0),vDraw,z1,tPen\WObj:=wPaper;
    MoveL Offs(pOrigin,74.0,13.5,0.0),vDraw,fine,tPen\WObj:=wPaper;
    MoveL Offs(pOrigin,74.0,13.5,15.0),vApproach,z5,tPen\WObj:=wPaper;
    MoveL Offs(pOrigin,74.0,14.8,15.0),vTravel,z5,tPen\WObj:=wPaper;
    MoveL Offs(pOrigin,74.0,14.8,0.0),vApproach,fine,tPen\WObj:=wPaper;
    MoveL Offs(pOrigin,73.8,15.0,0.0),vDraw,z1,tPen\WObj:=wPaper;
    MoveL Offs(pOrigin,74.0,15.2,0.0),vDraw,z1,tPen\WObj:=wPaper;
    MoveL Offs(pOrigin,74.9,15.2,0.0),vDraw,z1,tPen\WObj:=wPaper;
    MoveL Offs(pOrigin,75.1,15.0,0.0),vDraw,z1,tPen\WObj:=wPaper;
    MoveL Offs(pOrigin,74.9,14.8,0.0),vDraw,z1,tPen\WObj:=wPaper;
    MoveL Offs(pOrigin,74.0,14.8,0.0),vDraw,fine,tPen\WObj:=wPaper;
    MoveL Offs(pOrigin,74.0,14.8,15.0),vApproach,z5,tPen\WObj:=wPaper;
    MoveL Offs(pOrigin,75.5,14.8,15.0),vTravel,z5,tPen\WObj:=wPaper;
    MoveL Offs(pOrigin,75.5,14.8,0.0),vApproach,fine,tPen\WObj:=wPaper;
    MoveL Offs(pOrigin,75.7,15.0,0.0),vDraw,z1,tPen\WObj:=wPaper;
    MoveL Offs(pOrigin,77.0,15.0,0.0),vDraw,z1,tPen\WObj:=wPaper;
    MoveL Offs(pOrigin,77.2,14.8,0.0),vDraw,z1,tPen\WObj:=wPaper;
    MoveL Offs(pOrigin,77.0,14.6,0.0),vDraw,z1,tPen\WObj:=wPaper;
    MoveL Offs(pOrigin,75.7,14.6,0.0),vDraw,z1,tPen\WObj:=wPaper;
    MoveL Offs(pOrigin,75.5,14.8,0.0),vDraw,fine,tPen\WObj:=wPaper;
    MoveL Offs(pOrigin,75.5,14.8,15.0),vApproach,z5,tPen\WObj:=wPaper;
    MoveL Offs(pOrigin,75.9,13.7,15.0),vTravel,z5,tPen\WObj:=wPaper;
    MoveL Offs(pOrigin,75.9,13.7,0.0),vApproach,fine,tPen\WObj:=wPaper;
    MoveL Offs(pOrigin,76.6,13.7,0.0),vDraw,z1,tPen\WObj:=wPaper;
    MoveL Offs(pOrigin,76.8,13.5,0.0),vDraw,z1,tPen\WObj:=wPaper;
    MoveL Offs(pOrigin,76.6,13.3,0.0),vDraw,z1,tPen\WObj:=wPaper;
    MoveL Offs(pOrigin,75.9,13.3,0.0),vDraw,z1,tPen\WObj:=wPaper;
    MoveL Offs(pOrigin,75.7,13.5,0.0),vDraw,z1,tPen\WObj:=wPaper;
    MoveL Offs(pOrigin,75.9,13.7,0.0),vDraw,fine,tPen\WObj:=wPaper;
    MoveL Offs(pOrigin,75.9,13.7,15.0),vApproach,z5,tPen\WObj:=wPaper;
    MoveL Offs(pOrigin,75.7,12.9,15.0),vTravel,z5,tPen\WObj:=wPaper;
    MoveL Offs(pOrigin,75.7,12.9,0.0),vApproach,fine,tPen\WObj:=wPaper;
    MoveL Offs(pOrigin,77.0,12.9,0.0),vDraw,z1,tPen\WObj:=wPaper;
    MoveL Offs(pOrigin,77.2,12.7,0.0),vDraw,z1,tPen\WObj:=wPaper;
    MoveL Offs(pOrigin,77.0,12.6,0.0),vDraw,z1,tPen\WObj:=wPaper;
    MoveL Offs(pOrigin,75.7,12.6,0.0),vDraw,z1,tPen\WObj:=wPaper;
    MoveL Offs(pOrigin,75.5,12.7,0.0),vDraw,z1,tPen\WObj:=wPaper;
    MoveL Offs(pOrigin,75.7,12.9,0.0),vDraw,fine,tPen\WObj:=wPaper;
    MoveL Offs(pOrigin,75.7,12.9,15.0),vApproach,z5,tPen\WObj:=wPaper;
    MoveL Offs(pOrigin,77.4,12.6,15.0),vTravel,z5,tPen\WObj:=wPaper;
    MoveL Offs(pOrigin,77.4,12.6,0.0),vApproach,fine,tPen\WObj:=wPaper;
    MoveL Offs(pOrigin,77.6,12.7,0.0),vDraw,z1,tPen\WObj:=wPaper;
    MoveL Offs(pOrigin,78.9,12.7,0.0),vDraw,z1,tPen\WObj:=wPaper;
    MoveL Offs(pOrigin,79.1,12.6,0.0),vDraw,z1,tPen\WObj:=wPaper;
    MoveL Offs(pOrigin,78.9,12.4,0.0),vDraw,z1,tPen\WObj:=wPaper;
    MoveL Offs(pOrigin,77.6,12.4,0.0),vDraw,z1,tPen\WObj:=wPaper;
    MoveL Offs(pOrigin,77.4,12.6,0.0),vDraw,fine,tPen\WObj:=wPaper;
    MoveL Offs(pOrigin,77.4,12.6,15.0),vApproach,z5,tPen\WObj:=wPaper;
    MoveL Offs(pOrigin,77.6,13.1,15.0),vTravel,z5,tPen\WObj:=wPaper;
    MoveL Offs(pOrigin,77.6,13.1,0.0),vApproach,fine,tPen\WObj:=wPaper;
    MoveL Offs(pOrigin,77.4,13.3,0.0),vDraw,z1,tPen\WObj:=wPaper;
    MoveL Offs(pOrigin,77.6,13.5,0.0),vDraw,z1,tPen\WObj:=wPaper;
    MoveL Offs(pOrigin,78.5,13.5,0.0),vDraw,z1,tPen\WObj:=wPaper;
    MoveL Offs(pOrigin,78.7,13.3,0.0),vDraw,z1,tPen\WObj:=wPaper;
    MoveL Offs(pOrigin,78.5,13.1,0.0),vDraw,z1,tPen\WObj:=wPaper;
    MoveL Offs(pOrigin,77.6,13.1,0.0),vDraw,fine,tPen\WObj:=wPaper;
    MoveL Offs(pOrigin,77.6,13.1,15.0),vApproach,z5,tPen\WObj:=wPaper;
    MoveL Offs(pOrigin,77.6,14.4,15.0),vTravel,z5,tPen\WObj:=wPaper;
    MoveL Offs(pOrigin,77.6,14.4,0.0),vApproach,fine,tPen\WObj:=wPaper;
    MoveL Offs(pOrigin,77.4,14.6,0.0),vDraw,z1,tPen\WObj:=wPaper;
    MoveL Offs(pOrigin,77.6,14.8,0.0),vDraw,z1,tPen\WObj:=wPaper;
    MoveL Offs(pOrigin,79.1,14.8,0.0),vDraw,z1,tPen\WObj:=wPaper;
    MoveL Offs(pOrigin,79.3,14.6,0.0),vDraw,z1,tPen\WObj:=wPaper;
    MoveL Offs(pOrigin,79.1,14.4,0.0),vDraw,z1,tPen\WObj:=wPaper;
    MoveL Offs(pOrigin,77.6,14.4,0.0),vDraw,fine,tPen\WObj:=wPaper;
    MoveL Offs(pOrigin,77.6,14.4,15.0),vApproach,z5,tPen\WObj:=wPaper;
    MoveL Offs(pOrigin,79.1,14.4,15.0),vTravel,z5,tPen\WObj:=wPaper;
    MoveL Offs(pOrigin,79.1,14.4,0.0),vApproach,fine,tPen\WObj:=wPaper;
    MoveL Offs(pOrigin,79.3,14.6,0.0),vDraw,z1,tPen\WObj:=wPaper;
    MoveL Offs(pOrigin,81.0,14.6,0.0),vDraw,z1,tPen\WObj:=wPaper;
    MoveL Offs(pOrigin,81.2,14.4,0.0),vDraw,z1,tPen\WObj:=wPaper;
    MoveL Offs(pOrigin,81.0,14.3,0.0),vDraw,z1,tPen\WObj:=wPaper;
    MoveL Offs(pOrigin,79.3,14.3,0.0),vDraw,z1,tPen\WObj:=wPaper;
    MoveL Offs(pOrigin,79.1,14.4,0.0),vDraw,fine,tPen\WObj:=wPaper;
    MoveL Offs(pOrigin,79.1,14.4,15.0),vApproach,z5,tPen\WObj:=wPaper;
    MoveL Offs(pOrigin,79.5,13.3,15.0),vTravel,z5,tPen\WObj:=wPaper;
    MoveL Offs(pOrigin,79.5,13.3,0.0),vApproach,fine,tPen\WObj:=wPaper;
    MoveL Offs(pOrigin,80.4,13.3,0.0),vDraw,z1,tPen\WObj:=wPaper;
    MoveL Offs(pOrigin,80.6,13.1,0.0),vDraw,z1,tPen\WObj:=wPaper;
    MoveL Offs(pOrigin,80.4,12.9,0.0),vDraw,z1,tPen\WObj:=wPaper;
    MoveL Offs(pOrigin,79.5,12.9,0.0),vDraw,z1,tPen\WObj:=wPaper;
    MoveL Offs(pOrigin,79.3,13.1,0.0),vDraw,z1,tPen\WObj:=wPaper;
    MoveL Offs(pOrigin,79.5,13.3,0.0),vDraw,fine,tPen\WObj:=wPaper;
    MoveL Offs(pOrigin,79.5,13.3,15.0),vApproach,z5,tPen\WObj:=wPaper;
    MoveL Offs(pOrigin,79.3,12.6,15.0),vTravel,z5,tPen\WObj:=wPaper;
    MoveL Offs(pOrigin,79.3,12.6,0.0),vApproach,fine,tPen\WObj:=wPaper;
    MoveL Offs(pOrigin,80.6,12.6,0.0),vDraw,z1,tPen\WObj:=wPaper;
  ENDPROC

  PROC Part100()
    MoveL Offs(pOrigin,80.8,12.4,0.0),vDraw,z1,tPen\WObj:=wPaper;
    MoveL Offs(pOrigin,80.6,12.2,0.0),vDraw,z1,tPen\WObj:=wPaper;
    MoveL Offs(pOrigin,79.3,12.2,0.0),vDraw,z1,tPen\WObj:=wPaper;
    MoveL Offs(pOrigin,79.1,12.4,0.0),vDraw,z1,tPen\WObj:=wPaper;
    MoveL Offs(pOrigin,79.3,12.6,0.0),vDraw,fine,tPen\WObj:=wPaper;
    MoveL Offs(pOrigin,79.3,12.6,15.0),vApproach,z5,tPen\WObj:=wPaper;
    MoveL Offs(pOrigin,80.8,12.2,15.0),vTravel,z5,tPen\WObj:=wPaper;
    MoveL Offs(pOrigin,80.8,12.2,0.0),vApproach,fine,tPen\WObj:=wPaper;
    MoveL Offs(pOrigin,81.0,12.4,0.0),vDraw,z1,tPen\WObj:=wPaper;
    MoveL Offs(pOrigin,82.5,12.4,0.0),vDraw,z1,tPen\WObj:=wPaper;
    MoveL Offs(pOrigin,82.7,12.2,0.0),vDraw,z1,tPen\WObj:=wPaper;
    MoveL Offs(pOrigin,82.5,12.0,0.0),vDraw,z1,tPen\WObj:=wPaper;
    MoveL Offs(pOrigin,81.0,12.0,0.0),vDraw,z1,tPen\WObj:=wPaper;
    MoveL Offs(pOrigin,80.8,12.2,0.0),vDraw,fine,tPen\WObj:=wPaper;
    MoveL Offs(pOrigin,80.8,12.2,15.0),vApproach,z5,tPen\WObj:=wPaper;
    MoveL Offs(pOrigin,81.2,12.7,15.0),vTravel,z5,tPen\WObj:=wPaper;
    MoveL Offs(pOrigin,81.2,12.7,0.0),vApproach,fine,tPen\WObj:=wPaper;
    MoveL Offs(pOrigin,81.0,12.9,0.0),vDraw,z1,tPen\WObj:=wPaper;
    MoveL Offs(pOrigin,81.2,13.1,0.0),vDraw,z1,tPen\WObj:=wPaper;
    MoveL Offs(pOrigin,82.1,13.1,0.0),vDraw,z1,tPen\WObj:=wPaper;
    MoveL Offs(pOrigin,82.3,12.9,0.0),vDraw,z1,tPen\WObj:=wPaper;
    MoveL Offs(pOrigin,82.1,12.7,0.0),vDraw,z1,tPen\WObj:=wPaper;
    MoveL Offs(pOrigin,81.2,12.7,0.0),vDraw,fine,tPen\WObj:=wPaper;
    MoveL Offs(pOrigin,81.2,12.7,15.0),vApproach,z5,tPen\WObj:=wPaper;
    MoveL Offs(pOrigin,81.2,14.1,15.0),vTravel,z5,tPen\WObj:=wPaper;
    MoveL Offs(pOrigin,81.2,14.1,0.0),vApproach,fine,tPen\WObj:=wPaper;
    MoveL Offs(pOrigin,81.0,14.3,0.0),vDraw,z1,tPen\WObj:=wPaper;
    MoveL Offs(pOrigin,81.2,14.4,0.0),vDraw,z1,tPen\WObj:=wPaper;
    MoveL Offs(pOrigin,83.1,14.4,0.0),vDraw,z1,tPen\WObj:=wPaper;
    MoveL Offs(pOrigin,83.3,14.3,0.0),vDraw,z1,tPen\WObj:=wPaper;
    MoveL Offs(pOrigin,85.0,14.3,0.0),vDraw,z1,tPen\WObj:=wPaper;
    MoveL Offs(pOrigin,85.1,14.1,0.0),vDraw,z1,tPen\WObj:=wPaper;
    MoveL Offs(pOrigin,86.8,14.1,0.0),vDraw,z1,tPen\WObj:=wPaper;
    MoveL Offs(pOrigin,87.0,13.9,0.0),vDraw,z1,tPen\WObj:=wPaper;
    MoveL Offs(pOrigin,88.9,13.9,0.0),vDraw,z1,tPen\WObj:=wPaper;
    MoveL Offs(pOrigin,89.1,13.7,0.0),vDraw,z1,tPen\WObj:=wPaper;
    MoveL Offs(pOrigin,90.8,13.7,0.0),vDraw,z1,tPen\WObj:=wPaper;
    MoveL Offs(pOrigin,91.0,13.5,0.0),vDraw,z1,tPen\WObj:=wPaper;
    MoveL Offs(pOrigin,92.7,13.5,0.0),vDraw,z1,tPen\WObj:=wPaper;
    MoveL Offs(pOrigin,92.9,13.3,0.0),vDraw,z1,tPen\WObj:=wPaper;
    MoveL Offs(pOrigin,94.8,13.3,0.0),vDraw,z1,tPen\WObj:=wPaper;
    MoveL Offs(pOrigin,95.0,13.1,0.0),vDraw,z1,tPen\WObj:=wPaper;
    MoveL Offs(pOrigin,96.1,13.1,0.0),vDraw,z1,tPen\WObj:=wPaper;
    MoveL Offs(pOrigin,96.3,12.9,0.0),vDraw,z1,tPen\WObj:=wPaper;
    MoveL Offs(pOrigin,96.3,12.7,0.0),vDraw,z1,tPen\WObj:=wPaper;
    MoveL Offs(pOrigin,96.1,12.6,0.0),vDraw,z1,tPen\WObj:=wPaper;
    MoveL Offs(pOrigin,95.7,12.6,0.0),vDraw,z1,tPen\WObj:=wPaper;
    MoveL Offs(pOrigin,95.5,12.7,0.0),vDraw,z1,tPen\WObj:=wPaper;
    MoveL Offs(pOrigin,94.0,12.7,0.0),vDraw,z1,tPen\WObj:=wPaper;
    MoveL Offs(pOrigin,93.8,12.9,0.0),vDraw,z1,tPen\WObj:=wPaper;
    MoveL Offs(pOrigin,92.1,12.9,0.0),vDraw,z1,tPen\WObj:=wPaper;
    MoveL Offs(pOrigin,91.9,13.1,0.0),vDraw,z1,tPen\WObj:=wPaper;
    MoveL Offs(pOrigin,90.4,13.1,0.0),vDraw,z1,tPen\WObj:=wPaper;
    MoveL Offs(pOrigin,90.2,13.3,0.0),vDraw,z1,tPen\WObj:=wPaper;
    MoveL Offs(pOrigin,88.5,13.3,0.0),vDraw,z1,tPen\WObj:=wPaper;
    MoveL Offs(pOrigin,88.4,13.5,0.0),vDraw,z1,tPen\WObj:=wPaper;
    MoveL Offs(pOrigin,86.8,13.5,0.0),vDraw,z1,tPen\WObj:=wPaper;
    MoveL Offs(pOrigin,86.7,13.7,0.0),vDraw,z1,tPen\WObj:=wPaper;
    MoveL Offs(pOrigin,85.0,13.7,0.0),vDraw,z1,tPen\WObj:=wPaper;
    MoveL Offs(pOrigin,84.8,13.9,0.0),vDraw,z1,tPen\WObj:=wPaper;
    MoveL Offs(pOrigin,83.1,13.9,0.0),vDraw,z1,tPen\WObj:=wPaper;
    MoveL Offs(pOrigin,82.9,14.1,0.0),vDraw,z1,tPen\WObj:=wPaper;
    MoveL Offs(pOrigin,81.2,14.1,0.0),vDraw,fine,tPen\WObj:=wPaper;
    MoveL Offs(pOrigin,81.2,14.1,15.0),vApproach,z5,tPen\WObj:=wPaper;
    MoveL Offs(pOrigin,82.9,12.7,15.0),vTravel,z5,tPen\WObj:=wPaper;
    MoveL Offs(pOrigin,82.9,12.7,0.0),vApproach,fine,tPen\WObj:=wPaper;
    MoveL Offs(pOrigin,83.1,12.9,0.0),vDraw,z1,tPen\WObj:=wPaper;
    MoveL Offs(pOrigin,83.8,12.9,0.0),vDraw,z1,tPen\WObj:=wPaper;
    MoveL Offs(pOrigin,84.0,12.7,0.0),vDraw,z1,tPen\WObj:=wPaper;
    MoveL Offs(pOrigin,83.8,12.6,0.0),vDraw,z1,tPen\WObj:=wPaper;
    MoveL Offs(pOrigin,83.1,12.6,0.0),vDraw,z1,tPen\WObj:=wPaper;
    MoveL Offs(pOrigin,82.9,12.7,0.0),vDraw,fine,tPen\WObj:=wPaper;
    MoveL Offs(pOrigin,82.9,12.7,15.0),vApproach,z5,tPen\WObj:=wPaper;
    MoveL Offs(pOrigin,83.1,12.2,15.0),vTravel,z5,tPen\WObj:=wPaper;
    MoveL Offs(pOrigin,83.1,12.2,0.0),vApproach,fine,tPen\WObj:=wPaper;
    MoveL Offs(pOrigin,84.4,12.2,0.0),vDraw,z1,tPen\WObj:=wPaper;
    MoveL Offs(pOrigin,84.6,12.0,0.0),vDraw,z1,tPen\WObj:=wPaper;
    MoveL Offs(pOrigin,84.4,11.8,0.0),vDraw,z1,tPen\WObj:=wPaper;
    MoveL Offs(pOrigin,83.1,11.8,0.0),vDraw,z1,tPen\WObj:=wPaper;
    MoveL Offs(pOrigin,82.9,12.0,0.0),vDraw,z1,tPen\WObj:=wPaper;
    MoveL Offs(pOrigin,83.1,12.2,0.0),vDraw,fine,tPen\WObj:=wPaper;
    MoveL Offs(pOrigin,83.1,12.2,15.0),vApproach,z5,tPen\WObj:=wPaper;
    MoveL Offs(pOrigin,84.8,11.8,15.0),vTravel,z5,tPen\WObj:=wPaper;
    MoveL Offs(pOrigin,84.8,11.8,0.0),vApproach,fine,tPen\WObj:=wPaper;
    MoveL Offs(pOrigin,85.0,12.0,0.0),vDraw,z1,tPen\WObj:=wPaper;
    MoveL Offs(pOrigin,86.1,12.0,0.0),vDraw,z1,tPen\WObj:=wPaper;
    MoveL Offs(pOrigin,86.3,11.8,0.0),vDraw,z1,tPen\WObj:=wPaper;
    MoveL Offs(pOrigin,86.1,11.6,0.0),vDraw,z1,tPen\WObj:=wPaper;
    MoveL Offs(pOrigin,85.0,11.6,0.0),vDraw,z1,tPen\WObj:=wPaper;
    MoveL Offs(pOrigin,84.8,11.8,0.0),vDraw,fine,tPen\WObj:=wPaper;
    MoveL Offs(pOrigin,84.8,11.8,15.0),vApproach,z5,tPen\WObj:=wPaper;
    MoveL Offs(pOrigin,85.0,12.4,15.0),vTravel,z5,tPen\WObj:=wPaper;
    MoveL Offs(pOrigin,85.0,12.4,0.0),vApproach,fine,tPen\WObj:=wPaper;
    MoveL Offs(pOrigin,84.8,12.6,0.0),vDraw,z1,tPen\WObj:=wPaper;
    MoveL Offs(pOrigin,85.0,12.7,0.0),vDraw,z1,tPen\WObj:=wPaper;
    MoveL Offs(pOrigin,85.7,12.7,0.0),vDraw,z1,tPen\WObj:=wPaper;
    MoveL Offs(pOrigin,85.9,12.6,0.0),vDraw,z1,tPen\WObj:=wPaper;
    MoveL Offs(pOrigin,85.7,12.4,0.0),vDraw,z1,tPen\WObj:=wPaper;
    MoveL Offs(pOrigin,85.0,12.4,0.0),vDraw,fine,tPen\WObj:=wPaper;
    MoveL Offs(pOrigin,85.0,12.4,15.0),vApproach,z5,tPen\WObj:=wPaper;
    MoveL Offs(pOrigin,86.5,12.4,15.0),vTravel,z5,tPen\WObj:=wPaper;
    MoveL Offs(pOrigin,86.5,12.4,0.0),vApproach,fine,tPen\WObj:=wPaper;
    MoveL Offs(pOrigin,86.7,12.6,0.0),vDraw,z1,tPen\WObj:=wPaper;
    MoveL Offs(pOrigin,87.4,12.6,0.0),vDraw,z1,tPen\WObj:=wPaper;
    MoveL Offs(pOrigin,87.6,12.4,0.0),vDraw,z1,tPen\WObj:=wPaper;
    MoveL Offs(pOrigin,87.4,12.2,0.0),vDraw,z1,tPen\WObj:=wPaper;
    MoveL Offs(pOrigin,86.7,12.2,0.0),vDraw,z1,tPen\WObj:=wPaper;
    MoveL Offs(pOrigin,86.5,12.4,0.0),vDraw,fine,tPen\WObj:=wPaper;
    MoveL Offs(pOrigin,86.5,12.4,15.0),vApproach,z5,tPen\WObj:=wPaper;
    MoveL Offs(pOrigin,86.8,11.8,15.0),vTravel,z5,tPen\WObj:=wPaper;
    MoveL Offs(pOrigin,86.8,11.8,0.0),vApproach,fine,tPen\WObj:=wPaper;
    MoveL Offs(pOrigin,87.8,11.8,0.0),vDraw,z1,tPen\WObj:=wPaper;
    MoveL Offs(pOrigin,88.0,11.6,0.0),vDraw,z1,tPen\WObj:=wPaper;
    MoveL Offs(pOrigin,87.8,11.4,0.0),vDraw,z1,tPen\WObj:=wPaper;
    MoveL Offs(pOrigin,86.8,11.4,0.0),vDraw,z1,tPen\WObj:=wPaper;
    MoveL Offs(pOrigin,86.7,11.6,0.0),vDraw,z1,tPen\WObj:=wPaper;
    MoveL Offs(pOrigin,86.8,11.8,0.0),vDraw,fine,tPen\WObj:=wPaper;
    MoveL Offs(pOrigin,86.8,11.8,15.0),vApproach,z5,tPen\WObj:=wPaper;
    MoveL Offs(pOrigin,88.2,12.2,15.0),vTravel,z5,tPen\WObj:=wPaper;
    MoveL Offs(pOrigin,88.2,12.2,0.0),vApproach,fine,tPen\WObj:=wPaper;
  ENDPROC

  PROC Part101()
    MoveL Offs(pOrigin,88.4,12.4,0.0),vDraw,z1,tPen\WObj:=wPaper;
    MoveL Offs(pOrigin,89.3,12.4,0.0),vDraw,z1,tPen\WObj:=wPaper;
    MoveL Offs(pOrigin,89.5,12.2,0.0),vDraw,z1,tPen\WObj:=wPaper;
    MoveL Offs(pOrigin,89.3,12.0,0.0),vDraw,z1,tPen\WObj:=wPaper;
    MoveL Offs(pOrigin,88.4,12.0,0.0),vDraw,z1,tPen\WObj:=wPaper;
    MoveL Offs(pOrigin,88.2,12.2,0.0),vDraw,fine,tPen\WObj:=wPaper;
    MoveL Offs(pOrigin,88.2,12.2,15.0),vApproach,z5,tPen\WObj:=wPaper;
    MoveL Offs(pOrigin,88.5,11.6,15.0),vTravel,z5,tPen\WObj:=wPaper;
    MoveL Offs(pOrigin,88.5,11.6,0.0),vApproach,fine,tPen\WObj:=wPaper;
    MoveL Offs(pOrigin,89.7,11.6,0.0),vDraw,z1,tPen\WObj:=wPaper;
    MoveL Offs(pOrigin,89.9,11.4,0.0),vDraw,z1,tPen\WObj:=wPaper;
    MoveL Offs(pOrigin,89.7,11.2,0.0),vDraw,z1,tPen\WObj:=wPaper;
    MoveL Offs(pOrigin,88.5,11.2,0.0),vDraw,z1,tPen\WObj:=wPaper;
    MoveL Offs(pOrigin,88.4,11.4,0.0),vDraw,z1,tPen\WObj:=wPaper;
    MoveL Offs(pOrigin,88.5,11.6,0.0),vDraw,fine,tPen\WObj:=wPaper;
    MoveL Offs(pOrigin,88.5,11.6,15.0),vApproach,z5,tPen\WObj:=wPaper;
    MoveL Offs(pOrigin,90.1,11.2,15.0),vTravel,z5,tPen\WObj:=wPaper;
    MoveL Offs(pOrigin,90.1,11.2,0.0),vApproach,fine,tPen\WObj:=wPaper;
    MoveL Offs(pOrigin,90.2,11.4,0.0),vDraw,z1,tPen\WObj:=wPaper;
    MoveL Offs(pOrigin,91.6,11.4,0.0),vDraw,z1,tPen\WObj:=wPaper;
    MoveL Offs(pOrigin,91.8,11.2,0.0),vDraw,z1,tPen\WObj:=wPaper;
    MoveL Offs(pOrigin,91.6,11.0,0.0),vDraw,z1,tPen\WObj:=wPaper;
    MoveL Offs(pOrigin,90.2,11.0,0.0),vDraw,z1,tPen\WObj:=wPaper;
    MoveL Offs(pOrigin,90.1,11.2,0.0),vDraw,fine,tPen\WObj:=wPaper;
    MoveL Offs(pOrigin,90.1,11.2,15.0),vApproach,z5,tPen\WObj:=wPaper;
    MoveL Offs(pOrigin,90.2,11.8,15.0),vTravel,z5,tPen\WObj:=wPaper;
    MoveL Offs(pOrigin,90.2,11.8,0.0),vApproach,fine,tPen\WObj:=wPaper;
    MoveL Offs(pOrigin,90.1,12.0,0.0),vDraw,z1,tPen\WObj:=wPaper;
    MoveL Offs(pOrigin,90.2,12.2,0.0),vDraw,z1,tPen\WObj:=wPaper;
    MoveL Offs(pOrigin,91.0,12.2,0.0),vDraw,z1,tPen\WObj:=wPaper;
    MoveL Offs(pOrigin,91.2,12.0,0.0),vDraw,z1,tPen\WObj:=wPaper;
    MoveL Offs(pOrigin,91.0,11.8,0.0),vDraw,z1,tPen\WObj:=wPaper;
    MoveL Offs(pOrigin,90.2,11.8,0.0),vDraw,fine,tPen\WObj:=wPaper;
    MoveL Offs(pOrigin,90.2,11.8,15.0),vApproach,z5,tPen\WObj:=wPaper;
    MoveL Offs(pOrigin,91.9,11.8,15.0),vTravel,z5,tPen\WObj:=wPaper;
    MoveL Offs(pOrigin,91.9,11.8,0.0),vApproach,fine,tPen\WObj:=wPaper;
    MoveL Offs(pOrigin,92.1,12.0,0.0),vDraw,z1,tPen\WObj:=wPaper;
    MoveL Offs(pOrigin,92.9,12.0,0.0),vDraw,z1,tPen\WObj:=wPaper;
    MoveL Offs(pOrigin,93.1,11.8,0.0),vDraw,z1,tPen\WObj:=wPaper;
    MoveL Offs(pOrigin,92.9,11.6,0.0),vDraw,z1,tPen\WObj:=wPaper;
    MoveL Offs(pOrigin,92.1,11.6,0.0),vDraw,z1,tPen\WObj:=wPaper;
    MoveL Offs(pOrigin,91.9,11.8,0.0),vDraw,fine,tPen\WObj:=wPaper;
    MoveL Offs(pOrigin,91.9,11.8,15.0),vApproach,z5,tPen\WObj:=wPaper;
    MoveL Offs(pOrigin,92.1,11.2,15.0),vTravel,z5,tPen\WObj:=wPaper;
    MoveL Offs(pOrigin,92.1,11.2,0.0),vApproach,fine,tPen\WObj:=wPaper;
    MoveL Offs(pOrigin,93.3,11.2,0.0),vDraw,z1,tPen\WObj:=wPaper;
    MoveL Offs(pOrigin,93.5,11.0,0.0),vDraw,z1,tPen\WObj:=wPaper;
    MoveL Offs(pOrigin,93.3,10.9,0.0),vDraw,z1,tPen\WObj:=wPaper;
    MoveL Offs(pOrigin,92.1,10.9,0.0),vDraw,z1,tPen\WObj:=wPaper;
    MoveL Offs(pOrigin,91.9,11.0,0.0),vDraw,z1,tPen\WObj:=wPaper;
    MoveL Offs(pOrigin,92.1,11.2,0.0),vDraw,fine,tPen\WObj:=wPaper;
    MoveL Offs(pOrigin,92.1,11.2,15.0),vApproach,z5,tPen\WObj:=wPaper;
    MoveL Offs(pOrigin,93.6,10.9,15.0),vTravel,z5,tPen\WObj:=wPaper;
    MoveL Offs(pOrigin,93.6,10.9,0.0),vApproach,fine,tPen\WObj:=wPaper;
    MoveL Offs(pOrigin,93.8,11.0,0.0),vDraw,z1,tPen\WObj:=wPaper;
    MoveL Offs(pOrigin,95.2,11.0,0.0),vDraw,z1,tPen\WObj:=wPaper;
    MoveL Offs(pOrigin,95.3,10.9,0.0),vDraw,z1,tPen\WObj:=wPaper;
    MoveL Offs(pOrigin,95.2,10.7,0.0),vDraw,z1,tPen\WObj:=wPaper;
    MoveL Offs(pOrigin,93.8,10.7,0.0),vDraw,z1,tPen\WObj:=wPaper;
    MoveL Offs(pOrigin,93.6,10.9,0.0),vDraw,fine,tPen\WObj:=wPaper;
    MoveL Offs(pOrigin,93.6,10.9,15.0),vApproach,z5,tPen\WObj:=wPaper;
    MoveL Offs(pOrigin,93.8,11.4,15.0),vTravel,z5,tPen\WObj:=wPaper;
    MoveL Offs(pOrigin,93.8,11.4,0.0),vApproach,fine,tPen\WObj:=wPaper;
    MoveL Offs(pOrigin,93.6,11.6,0.0),vDraw,z1,tPen\WObj:=wPaper;
    MoveL Offs(pOrigin,93.8,11.8,0.0),vDraw,z1,tPen\WObj:=wPaper;
    MoveL Offs(pOrigin,94.6,11.8,0.0),vDraw,z1,tPen\WObj:=wPaper;
    MoveL Offs(pOrigin,94.8,11.6,0.0),vDraw,z1,tPen\WObj:=wPaper;
    MoveL Offs(pOrigin,94.6,11.4,0.0),vDraw,z1,tPen\WObj:=wPaper;
    MoveL Offs(pOrigin,93.8,11.4,0.0),vDraw,fine,tPen\WObj:=wPaper;
    MoveL Offs(pOrigin,93.8,11.4,15.0),vApproach,z5,tPen\WObj:=wPaper;
    MoveL Offs(pOrigin,95.5,10.7,15.0),vTravel,z5,tPen\WObj:=wPaper;
    MoveL Offs(pOrigin,95.5,10.7,0.0),vApproach,fine,tPen\WObj:=wPaper;
    MoveL Offs(pOrigin,95.7,10.9,0.0),vDraw,z1,tPen\WObj:=wPaper;
    MoveL Offs(pOrigin,96.5,10.9,0.0),vDraw,z1,tPen\WObj:=wPaper;
    MoveL Offs(pOrigin,96.7,11.0,0.0),vDraw,z1,tPen\WObj:=wPaper;
    MoveL Offs(pOrigin,96.7,11.8,0.0),vDraw,z1,tPen\WObj:=wPaper;
    MoveL Offs(pOrigin,96.5,12.0,0.0),vDraw,z1,tPen\WObj:=wPaper;
    MoveL Offs(pOrigin,96.9,12.4,0.0),vDraw,z1,tPen\WObj:=wPaper;
    MoveL Offs(pOrigin,97.0,12.2,0.0),vDraw,z1,tPen\WObj:=wPaper;
    MoveL Offs(pOrigin,97.0,10.7,0.0),vDraw,z1,tPen\WObj:=wPaper;
    MoveL Offs(pOrigin,96.9,10.5,0.0),vDraw,z1,tPen\WObj:=wPaper;
    MoveL Offs(pOrigin,95.7,10.5,0.0),vDraw,z1,tPen\WObj:=wPaper;
    MoveL Offs(pOrigin,95.5,10.7,0.0),vDraw,fine,tPen\WObj:=wPaper;
    MoveL Offs(pOrigin,95.5,10.7,15.0),vApproach,z5,tPen\WObj:=wPaper;
    MoveL Offs(pOrigin,98.0,10.7,15.0),vTravel,z5,tPen\WObj:=wPaper;
    MoveL Offs(pOrigin,98.0,10.7,0.0),vApproach,fine,tPen\WObj:=wPaper;
    MoveL Offs(pOrigin,98.2,10.9,0.0),vDraw,z1,tPen\WObj:=wPaper;
    MoveL Offs(pOrigin,99.3,10.9,0.0),vDraw,z1,tPen\WObj:=wPaper;
    MoveL Offs(pOrigin,99.5,10.7,0.0),vDraw,z1,tPen\WObj:=wPaper;
    MoveL Offs(pOrigin,99.3,10.5,0.0),vDraw,z1,tPen\WObj:=wPaper;
    MoveL Offs(pOrigin,98.2,10.5,0.0),vDraw,z1,tPen\WObj:=wPaper;
    MoveL Offs(pOrigin,98.0,10.7,0.0),vDraw,fine,tPen\WObj:=wPaper;
    MoveL Offs(pOrigin,98.0,10.7,15.0),vApproach,z5,tPen\WObj:=wPaper;
    MoveL Offs(pOrigin,98.6,10.1,15.0),vTravel,z5,tPen\WObj:=wPaper;
    MoveL Offs(pOrigin,98.6,10.1,0.0),vApproach,fine,tPen\WObj:=wPaper;
    MoveL Offs(pOrigin,99.3,10.1,0.0),vDraw,z1,tPen\WObj:=wPaper;
    MoveL Offs(pOrigin,99.5,9.9,0.0),vDraw,z1,tPen\WObj:=wPaper;
    MoveL Offs(pOrigin,99.3,9.7,0.0),vDraw,z1,tPen\WObj:=wPaper;
    MoveL Offs(pOrigin,98.6,9.7,0.0),vDraw,z1,tPen\WObj:=wPaper;
    MoveL Offs(pOrigin,98.4,9.9,0.0),vDraw,z1,tPen\WObj:=wPaper;
    MoveL Offs(pOrigin,98.6,10.1,0.0),vDraw,fine,tPen\WObj:=wPaper;
    MoveL Offs(pOrigin,98.6,10.1,15.0),vApproach,z5,tPen\WObj:=wPaper;
    MoveL Offs(pOrigin,98.7,11.2,15.0),vTravel,z5,tPen\WObj:=wPaper;
    MoveL Offs(pOrigin,98.7,11.2,0.0),vApproach,fine,tPen\WObj:=wPaper;
    MoveL Offs(pOrigin,98.4,11.6,0.0),vDraw,z1,tPen\WObj:=wPaper;
    MoveL Offs(pOrigin,98.4,12.0,0.0),vDraw,z1,tPen\WObj:=wPaper;
    MoveL Offs(pOrigin,98.7,12.4,0.0),vDraw,z1,tPen\WObj:=wPaper;
    MoveL Offs(pOrigin,98.7,12.6,0.0),vDraw,z1,tPen\WObj:=wPaper;
    MoveL Offs(pOrigin,98.9,12.7,0.0),vDraw,z1,tPen\WObj:=wPaper;
    MoveL Offs(pOrigin,98.9,13.1,0.0),vDraw,z1,tPen\WObj:=wPaper;
    MoveL Offs(pOrigin,99.1,13.3,0.0),vDraw,z1,tPen\WObj:=wPaper;
    MoveL Offs(pOrigin,100.4,13.3,0.0),vDraw,z1,tPen\WObj:=wPaper;
    MoveL Offs(pOrigin,100.6,13.1,0.0),vDraw,z1,tPen\WObj:=wPaper;
    MoveL Offs(pOrigin,102.5,13.1,0.0),vDraw,z1,tPen\WObj:=wPaper;
    MoveL Offs(pOrigin,102.7,12.9,0.0),vDraw,z1,tPen\WObj:=wPaper;
    MoveL Offs(pOrigin,103.1,12.9,0.0),vDraw,z1,tPen\WObj:=wPaper;
    MoveL Offs(pOrigin,103.3,12.7,0.0),vDraw,z1,tPen\WObj:=wPaper;
    MoveL Offs(pOrigin,102.9,12.2,0.0),vDraw,z1,tPen\WObj:=wPaper;
    MoveL Offs(pOrigin,102.9,11.4,0.0),vDraw,z1,tPen\WObj:=wPaper;
    MoveL Offs(pOrigin,102.7,11.2,0.0),vDraw,z1,tPen\WObj:=wPaper;
  ENDPROC

  PROC Part102()
    MoveL Offs(pOrigin,102.9,10.3,0.0),vDraw,z1,tPen\WObj:=wPaper;
    MoveL Offs(pOrigin,102.7,10.1,0.0),vDraw,z1,tPen\WObj:=wPaper;
    MoveL Offs(pOrigin,102.0,10.1,0.0),vDraw,z1,tPen\WObj:=wPaper;
    MoveL Offs(pOrigin,101.8,10.3,0.0),vDraw,z1,tPen\WObj:=wPaper;
    MoveL Offs(pOrigin,99.9,10.3,0.0),vDraw,z1,tPen\WObj:=wPaper;
    MoveL Offs(pOrigin,99.7,10.5,0.0),vDraw,z1,tPen\WObj:=wPaper;
    MoveL Offs(pOrigin,99.9,10.7,0.0),vDraw,z1,tPen\WObj:=wPaper;
    MoveL Offs(pOrigin,100.8,10.7,0.0),vDraw,z1,tPen\WObj:=wPaper;
    MoveL Offs(pOrigin,100.8,11.0,0.0),vDraw,z1,tPen\WObj:=wPaper;
    MoveL Offs(pOrigin,99.9,11.0,0.0),vDraw,z1,tPen\WObj:=wPaper;
    MoveL Offs(pOrigin,99.7,11.2,0.0),vDraw,z1,tPen\WObj:=wPaper;
    MoveL Offs(pOrigin,98.7,11.2,0.0),vDraw,fine,tPen\WObj:=wPaper;
    MoveL Offs(pOrigin,98.7,11.2,15.0),vApproach,z5,tPen\WObj:=wPaper;
    MoveL Offs(pOrigin,100.4,9.7,15.0),vTravel,z5,tPen\WObj:=wPaper;
    MoveL Offs(pOrigin,100.4,9.7,0.0),vApproach,fine,tPen\WObj:=wPaper;
    MoveL Offs(pOrigin,100.6,9.9,0.0),vDraw,z1,tPen\WObj:=wPaper;
    MoveL Offs(pOrigin,101.4,9.9,0.0),vDraw,z1,tPen\WObj:=wPaper;
    MoveL Offs(pOrigin,101.6,9.7,0.0),vDraw,z1,tPen\WObj:=wPaper;
    MoveL Offs(pOrigin,101.4,9.5,0.0),vDraw,z1,tPen\WObj:=wPaper;
    MoveL Offs(pOrigin,100.6,9.5,0.0),vDraw,z1,tPen\WObj:=wPaper;
    MoveL Offs(pOrigin,100.4,9.7,0.0),vDraw,fine,tPen\WObj:=wPaper;
    MoveL Offs(pOrigin,100.4,9.7,15.0),vApproach,z5,tPen\WObj:=wPaper;
    MoveL Offs(pOrigin,102.3,9.5,15.0),vTravel,z5,tPen\WObj:=wPaper;
    MoveL Offs(pOrigin,102.3,9.5,0.0),vApproach,fine,tPen\WObj:=wPaper;
    MoveL Offs(pOrigin,102.5,9.7,0.0),vDraw,z1,tPen\WObj:=wPaper;
    MoveL Offs(pOrigin,103.3,9.7,0.0),vDraw,z1,tPen\WObj:=wPaper;
    MoveL Offs(pOrigin,103.5,9.9,0.0),vDraw,z1,tPen\WObj:=wPaper;
    MoveL Offs(pOrigin,103.7,9.7,0.0),vDraw,z1,tPen\WObj:=wPaper;
    MoveL Offs(pOrigin,103.7,9.5,0.0),vDraw,z1,tPen\WObj:=wPaper;
    MoveL Offs(pOrigin,103.5,9.3,0.0),vDraw,z1,tPen\WObj:=wPaper;
    MoveL Offs(pOrigin,102.5,9.3,0.0),vDraw,z1,tPen\WObj:=wPaper;
    MoveL Offs(pOrigin,102.3,9.5,0.0),vDraw,fine,tPen\WObj:=wPaper;
    MoveL Offs(pOrigin,102.3,9.5,15.0),vApproach,z5,tPen\WObj:=wPaper;
    MoveL Offs(pOrigin,104.4,9.5,15.0),vTravel,z5,tPen\WObj:=wPaper;
    MoveL Offs(pOrigin,104.4,9.5,0.0),vApproach,fine,tPen\WObj:=wPaper;
    MoveL Offs(pOrigin,104.4,9.9,0.0),vDraw,z1,tPen\WObj:=wPaper;
    MoveL Offs(pOrigin,104.6,10.1,0.0),vDraw,z1,tPen\WObj:=wPaper;
    MoveL Offs(pOrigin,104.8,9.9,0.0),vDraw,z1,tPen\WObj:=wPaper;
    MoveL Offs(pOrigin,105.9,9.9,0.0),vDraw,z1,tPen\WObj:=wPaper;
    MoveL Offs(pOrigin,106.1,9.7,0.0),vDraw,z1,tPen\WObj:=wPaper;
    MoveL Offs(pOrigin,105.9,9.5,0.0),vDraw,z1,tPen\WObj:=wPaper;
    MoveL Offs(pOrigin,105.2,9.5,0.0),vDraw,z1,tPen\WObj:=wPaper;
    MoveL Offs(pOrigin,105.0,9.3,0.0),vDraw,z1,tPen\WObj:=wPaper;
    MoveL Offs(pOrigin,104.6,9.3,0.0),vDraw,z1,tPen\WObj:=wPaper;
    MoveL Offs(pOrigin,104.4,9.5,0.0),vDraw,fine,tPen\WObj:=wPaper;
    MoveL Offs(pOrigin,104.4,9.5,15.0),vApproach,z5,tPen\WObj:=wPaper;
    MoveL Offs(pOrigin,106.7,9.5,15.0),vTravel,z5,tPen\WObj:=wPaper;
    MoveL Offs(pOrigin,106.7,9.5,0.0),vApproach,fine,tPen\WObj:=wPaper;
    MoveL Offs(pOrigin,106.9,9.7,0.0),vDraw,z1,tPen\WObj:=wPaper;
    MoveL Offs(pOrigin,107.8,9.7,0.0),vDraw,z1,tPen\WObj:=wPaper;
    MoveL Offs(pOrigin,108.0,9.5,0.0),vDraw,z1,tPen\WObj:=wPaper;
    MoveL Offs(pOrigin,107.8,9.3,0.0),vDraw,z1,tPen\WObj:=wPaper;
    MoveL Offs(pOrigin,106.9,9.3,0.0),vDraw,z1,tPen\WObj:=wPaper;
    MoveL Offs(pOrigin,106.7,9.5,0.0),vDraw,fine,tPen\WObj:=wPaper;
    MoveL Offs(pOrigin,106.7,9.5,15.0),vApproach,z5,tPen\WObj:=wPaper;
    MoveL Offs(pOrigin,108.4,9.3,15.0),vTravel,z5,tPen\WObj:=wPaper;
    MoveL Offs(pOrigin,108.4,9.3,0.0),vApproach,fine,tPen\WObj:=wPaper;
    MoveL Offs(pOrigin,108.6,9.5,0.0),vDraw,z1,tPen\WObj:=wPaper;
    MoveL Offs(pOrigin,109.5,9.5,0.0),vDraw,z1,tPen\WObj:=wPaper;
    MoveL Offs(pOrigin,109.7,9.3,0.0),vDraw,z1,tPen\WObj:=wPaper;
    MoveL Offs(pOrigin,109.5,9.2,0.0),vDraw,z1,tPen\WObj:=wPaper;
    MoveL Offs(pOrigin,108.6,9.2,0.0),vDraw,z1,tPen\WObj:=wPaper;
    MoveL Offs(pOrigin,108.4,9.3,0.0),vDraw,fine,tPen\WObj:=wPaper;
    MoveL Offs(pOrigin,108.4,9.3,15.0),vApproach,z5,tPen\WObj:=wPaper;
    MoveL Offs(pOrigin,109.9,9.9,15.0),vTravel,z5,tPen\WObj:=wPaper;
    MoveL Offs(pOrigin,109.9,9.9,0.0),vApproach,fine,tPen\WObj:=wPaper;
    MoveL Offs(pOrigin,110.1,10.1,0.0),vDraw,z1,tPen\WObj:=wPaper;
    MoveL Offs(pOrigin,111.0,10.1,0.0),vDraw,z1,tPen\WObj:=wPaper;
    MoveL Offs(pOrigin,111.2,9.9,0.0),vDraw,z1,tPen\WObj:=wPaper;
    MoveL Offs(pOrigin,111.0,9.7,0.0),vDraw,z1,tPen\WObj:=wPaper;
    MoveL Offs(pOrigin,110.1,9.7,0.0),vDraw,z1,tPen\WObj:=wPaper;
    MoveL Offs(pOrigin,109.9,9.9,0.0),vDraw,fine,tPen\WObj:=wPaper;
    MoveL Offs(pOrigin,109.9,9.9,15.0),vApproach,z5,tPen\WObj:=wPaper;
    MoveL Offs(pOrigin,110.3,9.3,15.0),vTravel,z5,tPen\WObj:=wPaper;
    MoveL Offs(pOrigin,110.3,9.3,0.0),vApproach,fine,tPen\WObj:=wPaper;
    MoveL Offs(pOrigin,111.4,9.3,0.0),vDraw,z1,tPen\WObj:=wPaper;
    MoveL Offs(pOrigin,111.6,9.2,0.0),vDraw,z1,tPen\WObj:=wPaper;
    MoveL Offs(pOrigin,111.4,9.0,0.0),vDraw,z1,tPen\WObj:=wPaper;
    MoveL Offs(pOrigin,110.3,9.0,0.0),vDraw,z1,tPen\WObj:=wPaper;
    MoveL Offs(pOrigin,110.1,9.2,0.0),vDraw,z1,tPen\WObj:=wPaper;
    MoveL Offs(pOrigin,110.3,9.3,0.0),vDraw,fine,tPen\WObj:=wPaper;
    MoveL Offs(pOrigin,110.3,9.3,15.0),vApproach,z5,tPen\WObj:=wPaper;
    MoveL Offs(pOrigin,111.8,9.7,15.0),vTravel,z5,tPen\WObj:=wPaper;
    MoveL Offs(pOrigin,111.8,9.7,0.0),vApproach,fine,tPen\WObj:=wPaper;
    MoveL Offs(pOrigin,112.0,9.9,0.0),vDraw,z1,tPen\WObj:=wPaper;
    MoveL Offs(pOrigin,112.9,9.9,0.0),vDraw,z1,tPen\WObj:=wPaper;
    MoveL Offs(pOrigin,113.1,9.7,0.0),vDraw,z1,tPen\WObj:=wPaper;
    MoveL Offs(pOrigin,112.9,9.5,0.0),vDraw,z1,tPen\WObj:=wPaper;
    MoveL Offs(pOrigin,112.0,9.5,0.0),vDraw,z1,tPen\WObj:=wPaper;
    MoveL Offs(pOrigin,111.8,9.7,0.0),vDraw,fine,tPen\WObj:=wPaper;
    MoveL Offs(pOrigin,111.8,9.7,15.0),vApproach,z5,tPen\WObj:=wPaper;
    MoveL Offs(pOrigin,112.2,9.2,15.0),vTravel,z5,tPen\WObj:=wPaper;
    MoveL Offs(pOrigin,112.2,9.2,0.0),vApproach,fine,tPen\WObj:=wPaper;
    MoveL Offs(pOrigin,113.5,9.2,0.0),vDraw,z1,tPen\WObj:=wPaper;
    MoveL Offs(pOrigin,113.7,9.0,0.0),vDraw,z1,tPen\WObj:=wPaper;
    MoveL Offs(pOrigin,113.5,8.8,0.0),vDraw,z1,tPen\WObj:=wPaper;
    MoveL Offs(pOrigin,112.2,8.8,0.0),vDraw,z1,tPen\WObj:=wPaper;
    MoveL Offs(pOrigin,112.0,9.0,0.0),vDraw,z1,tPen\WObj:=wPaper;
    MoveL Offs(pOrigin,112.2,9.2,0.0),vDraw,fine,tPen\WObj:=wPaper;
    MoveL Offs(pOrigin,112.2,9.2,15.0),vApproach,z5,tPen\WObj:=wPaper;
    MoveL Offs(pOrigin,111.8,10.9,15.0),vTravel,z5,tPen\WObj:=wPaper;
    MoveL Offs(pOrigin,111.8,10.9,0.0),vApproach,fine,tPen\WObj:=wPaper;
    MoveL Offs(pOrigin,111.6,11.0,0.0),vDraw,z1,tPen\WObj:=wPaper;
    MoveL Offs(pOrigin,109.9,11.0,0.0),vDraw,z1,tPen\WObj:=wPaper;
    MoveL Offs(pOrigin,109.7,11.2,0.0),vDraw,z1,tPen\WObj:=wPaper;
    MoveL Offs(pOrigin,108.0,11.2,0.0),vDraw,z1,tPen\WObj:=wPaper;
    MoveL Offs(pOrigin,107.8,11.4,0.0),vDraw,z1,tPen\WObj:=wPaper;
    MoveL Offs(pOrigin,105.9,11.4,0.0),vDraw,z1,tPen\WObj:=wPaper;
    MoveL Offs(pOrigin,105.7,11.6,0.0),vDraw,z1,tPen\WObj:=wPaper;
    MoveL Offs(pOrigin,105.4,11.6,0.0),vDraw,z1,tPen\WObj:=wPaper;
    MoveL Offs(pOrigin,105.2,11.8,0.0),vDraw,z1,tPen\WObj:=wPaper;
    MoveL Offs(pOrigin,105.4,12.0,0.0),vDraw,z1,tPen\WObj:=wPaper;
    MoveL Offs(pOrigin,106.9,12.0,0.0),vDraw,z1,tPen\WObj:=wPaper;
    MoveL Offs(pOrigin,107.1,11.8,0.0),vDraw,z1,tPen\WObj:=wPaper;
    MoveL Offs(pOrigin,108.8,11.8,0.0),vDraw,z1,tPen\WObj:=wPaper;
    MoveL Offs(pOrigin,108.9,11.6,0.0),vDraw,z1,tPen\WObj:=wPaper;
    MoveL Offs(pOrigin,110.6,11.6,0.0),vDraw,z1,tPen\WObj:=wPaper;
    MoveL Offs(pOrigin,110.8,11.4,0.0),vDraw,z1,tPen\WObj:=wPaper;
    MoveL Offs(pOrigin,112.5,11.4,0.0),vDraw,z1,tPen\WObj:=wPaper;
    MoveL Offs(pOrigin,112.7,11.2,0.0),vDraw,z1,tPen\WObj:=wPaper;
  ENDPROC

  PROC Part103()
    MoveL Offs(pOrigin,114.4,11.2,0.0),vDraw,z1,tPen\WObj:=wPaper;
    MoveL Offs(pOrigin,114.6,11.0,0.0),vDraw,z1,tPen\WObj:=wPaper;
    MoveL Offs(pOrigin,117.4,11.0,0.0),vDraw,z1,tPen\WObj:=wPaper;
    MoveL Offs(pOrigin,117.6,10.9,0.0),vDraw,z1,tPen\WObj:=wPaper;
    MoveL Offs(pOrigin,117.4,10.7,0.0),vDraw,z1,tPen\WObj:=wPaper;
    MoveL Offs(pOrigin,116.9,10.7,0.0),vDraw,z1,tPen\WObj:=wPaper;
    MoveL Offs(pOrigin,116.7,10.5,0.0),vDraw,z1,tPen\WObj:=wPaper;
    MoveL Offs(pOrigin,115.6,10.5,0.0),vDraw,z1,tPen\WObj:=wPaper;
    MoveL Offs(pOrigin,115.4,10.7,0.0),vDraw,z1,tPen\WObj:=wPaper;
    MoveL Offs(pOrigin,113.7,10.7,0.0),vDraw,z1,tPen\WObj:=wPaper;
    MoveL Offs(pOrigin,113.5,10.9,0.0),vDraw,z1,tPen\WObj:=wPaper;
    MoveL Offs(pOrigin,111.8,10.9,0.0),vDraw,fine,tPen\WObj:=wPaper;
    MoveL Offs(pOrigin,111.8,10.9,15.0),vApproach,z5,tPen\WObj:=wPaper;
    MoveL Offs(pOrigin,112.0,12.4,15.0),vTravel,z5,tPen\WObj:=wPaper;
    MoveL Offs(pOrigin,112.0,12.4,0.0),vApproach,fine,tPen\WObj:=wPaper;
    MoveL Offs(pOrigin,111.8,12.6,0.0),vDraw,z1,tPen\WObj:=wPaper;
    MoveL Offs(pOrigin,110.1,12.6,0.0),vDraw,z1,tPen\WObj:=wPaper;
    MoveL Offs(pOrigin,109.9,12.7,0.0),vDraw,z1,tPen\WObj:=wPaper;
    MoveL Offs(pOrigin,108.4,12.7,0.0),vDraw,z1,tPen\WObj:=wPaper;
    MoveL Offs(pOrigin,108.2,12.9,0.0),vDraw,z1,tPen\WObj:=wPaper;
    MoveL Offs(pOrigin,108.4,13.1,0.0),vDraw,z1,tPen\WObj:=wPaper;
    MoveL Offs(pOrigin,108.9,13.1,0.0),vDraw,z1,tPen\WObj:=wPaper;
    MoveL Offs(pOrigin,109.1,13.3,0.0),vDraw,z1,tPen\WObj:=wPaper;
    MoveL Offs(pOrigin,109.9,13.3,0.0),vDraw,z1,tPen\WObj:=wPaper;
    MoveL Offs(pOrigin,110.1,13.5,0.0),vDraw,z1,tPen\WObj:=wPaper;
    MoveL Offs(pOrigin,110.6,13.5,0.0),vDraw,z1,tPen\WObj:=wPaper;
    MoveL Offs(pOrigin,110.8,13.7,0.0),vDraw,z1,tPen\WObj:=wPaper;
    MoveL Offs(pOrigin,111.6,13.7,0.0),vDraw,z1,tPen\WObj:=wPaper;
    MoveL Offs(pOrigin,111.8,13.9,0.0),vDraw,z1,tPen\WObj:=wPaper;
    MoveL Offs(pOrigin,112.5,13.9,0.0),vDraw,z1,tPen\WObj:=wPaper;
    MoveL Offs(pOrigin,112.7,14.1,0.0),vDraw,z1,tPen\WObj:=wPaper;
    MoveL Offs(pOrigin,113.3,14.1,0.0),vDraw,z1,tPen\WObj:=wPaper;
    MoveL Offs(pOrigin,113.5,14.3,0.0),vDraw,z1,tPen\WObj:=wPaper;
    MoveL Offs(pOrigin,114.2,14.3,0.0),vDraw,z1,tPen\WObj:=wPaper;
    MoveL Offs(pOrigin,114.4,14.4,0.0),vDraw,z1,tPen\WObj:=wPaper;
    MoveL Offs(pOrigin,115.2,14.4,0.0),vDraw,z1,tPen\WObj:=wPaper;
    MoveL Offs(pOrigin,115.4,14.6,0.0),vDraw,z1,tPen\WObj:=wPaper;
    MoveL Offs(pOrigin,115.9,14.6,0.0),vDraw,z1,tPen\WObj:=wPaper;
    MoveL Offs(pOrigin,116.1,14.8,0.0),vDraw,z1,tPen\WObj:=wPaper;
    MoveL Offs(pOrigin,116.9,14.8,0.0),vDraw,z1,tPen\WObj:=wPaper;
    MoveL Offs(pOrigin,117.1,15.0,0.0),vDraw,z1,tPen\WObj:=wPaper;
    MoveL Offs(pOrigin,117.6,15.0,0.0),vDraw,z1,tPen\WObj:=wPaper;
    MoveL Offs(pOrigin,117.8,15.2,0.0),vDraw,z1,tPen\WObj:=wPaper;
    MoveL Offs(pOrigin,118.6,15.2,0.0),vDraw,z1,tPen\WObj:=wPaper;
    MoveL Offs(pOrigin,118.8,15.4,0.0),vDraw,z1,tPen\WObj:=wPaper;
    MoveL Offs(pOrigin,119.5,15.4,0.0),vDraw,z1,tPen\WObj:=wPaper;
    MoveL Offs(pOrigin,119.7,15.6,0.0),vDraw,z1,tPen\WObj:=wPaper;
    MoveL Offs(pOrigin,120.3,15.6,0.0),vDraw,z1,tPen\WObj:=wPaper;
    MoveL Offs(pOrigin,120.5,15.8,0.0),vDraw,z1,tPen\WObj:=wPaper;
    MoveL Offs(pOrigin,121.2,15.8,0.0),vDraw,z1,tPen\WObj:=wPaper;
    MoveL Offs(pOrigin,121.4,16.0,0.0),vDraw,z1,tPen\WObj:=wPaper;
    MoveL Offs(pOrigin,122.2,16.0,0.0),vDraw,z1,tPen\WObj:=wPaper;
    MoveL Offs(pOrigin,122.4,16.1,0.0),vDraw,z1,tPen\WObj:=wPaper;
    MoveL Offs(pOrigin,123.1,16.1,0.0),vDraw,z1,tPen\WObj:=wPaper;
    MoveL Offs(pOrigin,123.3,16.3,0.0),vDraw,z1,tPen\WObj:=wPaper;
    MoveL Offs(pOrigin,124.1,16.3,0.0),vDraw,z1,tPen\WObj:=wPaper;
    MoveL Offs(pOrigin,124.2,16.5,0.0),vDraw,z1,tPen\WObj:=wPaper;
    MoveL Offs(pOrigin,124.8,16.5,0.0),vDraw,z1,tPen\WObj:=wPaper;
    MoveL Offs(pOrigin,125.0,16.7,0.0),vDraw,z1,tPen\WObj:=wPaper;
    MoveL Offs(pOrigin,125.6,16.7,0.0),vDraw,z1,tPen\WObj:=wPaper;
    MoveL Offs(pOrigin,125.8,16.9,0.0),vDraw,z1,tPen\WObj:=wPaper;
    MoveL Offs(pOrigin,126.7,16.9,0.0),vDraw,z1,tPen\WObj:=wPaper;
    MoveL Offs(pOrigin,126.9,17.1,0.0),vDraw,z1,tPen\WObj:=wPaper;
    MoveL Offs(pOrigin,127.3,16.7,0.0),vDraw,z1,tPen\WObj:=wPaper;
    MoveL Offs(pOrigin,127.5,16.7,0.0),vDraw,z1,tPen\WObj:=wPaper;
    MoveL Offs(pOrigin,128.0,16.3,0.0),vDraw,z1,tPen\WObj:=wPaper;
    MoveL Offs(pOrigin,128.8,16.3,0.0),vDraw,z1,tPen\WObj:=wPaper;
    MoveL Offs(pOrigin,129.0,16.1,0.0),vDraw,z1,tPen\WObj:=wPaper;
    MoveL Offs(pOrigin,132.2,16.1,0.0),vDraw,z1,tPen\WObj:=wPaper;
    MoveL Offs(pOrigin,132.4,16.0,0.0),vDraw,z1,tPen\WObj:=wPaper;
    MoveL Offs(pOrigin,132.2,15.8,0.0),vDraw,z1,tPen\WObj:=wPaper;
    MoveL Offs(pOrigin,131.6,15.8,0.0),vDraw,z1,tPen\WObj:=wPaper;
    MoveL Offs(pOrigin,131.4,15.6,0.0),vDraw,z1,tPen\WObj:=wPaper;
    MoveL Offs(pOrigin,130.9,15.6,0.0),vDraw,z1,tPen\WObj:=wPaper;
    MoveL Offs(pOrigin,130.7,15.4,0.0),vDraw,z1,tPen\WObj:=wPaper;
    MoveL Offs(pOrigin,130.1,15.4,0.0),vDraw,z1,tPen\WObj:=wPaper;
    MoveL Offs(pOrigin,129.9,15.2,0.0),vDraw,z1,tPen\WObj:=wPaper;
    MoveL Offs(pOrigin,129.3,15.2,0.0),vDraw,z1,tPen\WObj:=wPaper;
    MoveL Offs(pOrigin,129.2,15.0,0.0),vDraw,z1,tPen\WObj:=wPaper;
    MoveL Offs(pOrigin,128.6,15.0,0.0),vDraw,z1,tPen\WObj:=wPaper;
    MoveL Offs(pOrigin,128.4,14.8,0.0),vDraw,z1,tPen\WObj:=wPaper;
    MoveL Offs(pOrigin,127.8,14.8,0.0),vDraw,z1,tPen\WObj:=wPaper;
    MoveL Offs(pOrigin,127.6,14.6,0.0),vDraw,z1,tPen\WObj:=wPaper;
    MoveL Offs(pOrigin,127.1,14.6,0.0),vDraw,z1,tPen\WObj:=wPaper;
    MoveL Offs(pOrigin,126.9,14.4,0.0),vDraw,z1,tPen\WObj:=wPaper;
    MoveL Offs(pOrigin,126.5,14.4,0.0),vDraw,z1,tPen\WObj:=wPaper;
    MoveL Offs(pOrigin,126.3,14.3,0.0),vDraw,z1,tPen\WObj:=wPaper;
    MoveL Offs(pOrigin,125.8,14.3,0.0),vDraw,z1,tPen\WObj:=wPaper;
    MoveL Offs(pOrigin,125.6,14.1,0.0),vDraw,z1,tPen\WObj:=wPaper;
    MoveL Offs(pOrigin,125.0,14.1,0.0),vDraw,z1,tPen\WObj:=wPaper;
    MoveL Offs(pOrigin,124.8,13.9,0.0),vDraw,z1,tPen\WObj:=wPaper;
    MoveL Offs(pOrigin,124.2,13.9,0.0),vDraw,z1,tPen\WObj:=wPaper;
    MoveL Offs(pOrigin,124.1,13.7,0.0),vDraw,z1,tPen\WObj:=wPaper;
    MoveL Offs(pOrigin,123.5,13.7,0.0),vDraw,z1,tPen\WObj:=wPaper;
    MoveL Offs(pOrigin,123.3,13.5,0.0),vDraw,z1,tPen\WObj:=wPaper;
    MoveL Offs(pOrigin,122.7,13.5,0.0),vDraw,z1,tPen\WObj:=wPaper;
    MoveL Offs(pOrigin,122.5,13.3,0.0),vDraw,z1,tPen\WObj:=wPaper;
    MoveL Offs(pOrigin,122.0,13.3,0.0),vDraw,z1,tPen\WObj:=wPaper;
    MoveL Offs(pOrigin,121.8,13.1,0.0),vDraw,z1,tPen\WObj:=wPaper;
    MoveL Offs(pOrigin,121.2,13.1,0.0),vDraw,z1,tPen\WObj:=wPaper;
    MoveL Offs(pOrigin,121.0,12.9,0.0),vDraw,z1,tPen\WObj:=wPaper;
    MoveL Offs(pOrigin,120.5,12.9,0.0),vDraw,z1,tPen\WObj:=wPaper;
    MoveL Offs(pOrigin,120.3,12.7,0.0),vDraw,z1,tPen\WObj:=wPaper;
    MoveL Offs(pOrigin,119.7,12.7,0.0),vDraw,z1,tPen\WObj:=wPaper;
    MoveL Offs(pOrigin,119.5,12.6,0.0),vDraw,z1,tPen\WObj:=wPaper;
    MoveL Offs(pOrigin,119.0,12.6,0.0),vDraw,z1,tPen\WObj:=wPaper;
    MoveL Offs(pOrigin,118.8,12.4,0.0),vDraw,z1,tPen\WObj:=wPaper;
    MoveL Offs(pOrigin,118.0,12.4,0.0),vDraw,z1,tPen\WObj:=wPaper;
    MoveL Offs(pOrigin,117.8,12.2,0.0),vDraw,z1,tPen\WObj:=wPaper;
    MoveL Offs(pOrigin,117.3,12.2,0.0),vDraw,z1,tPen\WObj:=wPaper;
    MoveL Offs(pOrigin,117.1,12.0,0.0),vDraw,z1,tPen\WObj:=wPaper;
    MoveL Offs(pOrigin,115.6,12.0,0.0),vDraw,z1,tPen\WObj:=wPaper;
    MoveL Offs(pOrigin,115.4,12.2,0.0),vDraw,z1,tPen\WObj:=wPaper;
    MoveL Offs(pOrigin,113.7,12.2,0.0),vDraw,z1,tPen\WObj:=wPaper;
    MoveL Offs(pOrigin,113.5,12.4,0.0),vDraw,z1,tPen\WObj:=wPaper;
    MoveL Offs(pOrigin,112.0,12.4,0.0),vDraw,fine,tPen\WObj:=wPaper;
    MoveL Offs(pOrigin,112.0,12.4,15.0),vApproach,z5,tPen\WObj:=wPaper;
    MoveL Offs(pOrigin,114.0,9.7,15.0),vTravel,z5,tPen\WObj:=wPaper;
    MoveL Offs(pOrigin,114.0,9.7,0.0),vApproach,fine,tPen\WObj:=wPaper;
    MoveL Offs(pOrigin,114.8,9.7,0.0),vDraw,z1,tPen\WObj:=wPaper;
  ENDPROC

  PROC Part104()
    MoveL Offs(pOrigin,115.0,9.5,0.0),vDraw,z1,tPen\WObj:=wPaper;
    MoveL Offs(pOrigin,114.8,9.3,0.0),vDraw,z1,tPen\WObj:=wPaper;
    MoveL Offs(pOrigin,114.0,9.3,0.0),vDraw,z1,tPen\WObj:=wPaper;
    MoveL Offs(pOrigin,113.9,9.5,0.0),vDraw,z1,tPen\WObj:=wPaper;
    MoveL Offs(pOrigin,114.0,9.7,0.0),vDraw,fine,tPen\WObj:=wPaper;
    MoveL Offs(pOrigin,114.0,9.7,15.0),vApproach,z5,tPen\WObj:=wPaper;
    MoveL Offs(pOrigin,114.0,9.0,15.0),vTravel,z5,tPen\WObj:=wPaper;
    MoveL Offs(pOrigin,114.0,9.0,0.0),vApproach,fine,tPen\WObj:=wPaper;
    MoveL Offs(pOrigin,115.6,9.0,0.0),vDraw,z1,tPen\WObj:=wPaper;
    MoveL Offs(pOrigin,115.7,8.8,0.0),vDraw,z1,tPen\WObj:=wPaper;
    MoveL Offs(pOrigin,115.6,8.6,0.0),vDraw,z1,tPen\WObj:=wPaper;
    MoveL Offs(pOrigin,114.0,8.6,0.0),vDraw,z1,tPen\WObj:=wPaper;
    MoveL Offs(pOrigin,113.9,8.8,0.0),vDraw,z1,tPen\WObj:=wPaper;
    MoveL Offs(pOrigin,114.0,9.0,0.0),vDraw,fine,tPen\WObj:=wPaper;
    MoveL Offs(pOrigin,114.0,9.0,15.0),vApproach,z5,tPen\WObj:=wPaper;
    MoveL Offs(pOrigin,105.9,12.7,15.0),vTravel,z5,tPen\WObj:=wPaper;
    MoveL Offs(pOrigin,105.9,12.7,0.0),vApproach,fine,tPen\WObj:=wPaper;
    MoveL Offs(pOrigin,105.7,12.6,0.0),vDraw,z1,tPen\WObj:=wPaper;
    MoveL Offs(pOrigin,105.4,12.6,0.0),vDraw,z1,tPen\WObj:=wPaper;
    MoveL Offs(pOrigin,105.2,12.4,0.0),vDraw,z1,tPen\WObj:=wPaper;
    MoveL Offs(pOrigin,105.0,12.4,0.0),vDraw,z1,tPen\WObj:=wPaper;
    MoveL Offs(pOrigin,104.8,12.6,0.0),vDraw,z1,tPen\WObj:=wPaper;
    MoveL Offs(pOrigin,104.8,13.1,0.0),vDraw,z1,tPen\WObj:=wPaper;
    MoveL Offs(pOrigin,104.2,13.1,0.0),vDraw,z1,tPen\WObj:=wPaper;
    MoveL Offs(pOrigin,104.0,13.3,0.0),vDraw,z1,tPen\WObj:=wPaper;
    MoveL Offs(pOrigin,104.2,13.5,0.0),vDraw,z1,tPen\WObj:=wPaper;
    MoveL Offs(pOrigin,105.0,13.5,0.0),vDraw,z1,tPen\WObj:=wPaper;
    MoveL Offs(pOrigin,105.4,13.1,0.0),vDraw,z1,tPen\WObj:=wPaper;
    MoveL Offs(pOrigin,105.7,13.1,0.0),vDraw,z1,tPen\WObj:=wPaper;
    MoveL Offs(pOrigin,105.9,12.9,0.0),vDraw,z1,tPen\WObj:=wPaper;
    MoveL Offs(pOrigin,105.9,12.7,0.0),vDraw,fine,tPen\WObj:=wPaper;
    MoveL Offs(pOrigin,105.9,12.7,15.0),vApproach,z5,tPen\WObj:=wPaper;
    MoveL Offs(pOrigin,104.2,13.5,15.0),vTravel,z5,tPen\WObj:=wPaper;
    MoveL Offs(pOrigin,104.2,13.5,0.0),vApproach,fine,tPen\WObj:=wPaper;
    MoveL Offs(pOrigin,104.0,13.3,0.0),vDraw,z1,tPen\WObj:=wPaper;
    MoveL Offs(pOrigin,103.1,13.3,0.0),vDraw,z1,tPen\WObj:=wPaper;
    MoveL Offs(pOrigin,102.9,13.5,0.0),vDraw,z1,tPen\WObj:=wPaper;
    MoveL Offs(pOrigin,103.1,13.7,0.0),vDraw,z1,tPen\WObj:=wPaper;
    MoveL Offs(pOrigin,104.0,13.7,0.0),vDraw,z1,tPen\WObj:=wPaper;
    MoveL Offs(pOrigin,104.2,13.5,0.0),vDraw,fine,tPen\WObj:=wPaper;
    MoveL Offs(pOrigin,104.2,13.5,15.0),vApproach,z5,tPen\WObj:=wPaper;
    MoveL Offs(pOrigin,102.3,13.7,15.0),vTravel,z5,tPen\WObj:=wPaper;
    MoveL Offs(pOrigin,102.3,13.7,0.0),vApproach,fine,tPen\WObj:=wPaper;
    MoveL Offs(pOrigin,102.1,13.5,0.0),vDraw,z1,tPen\WObj:=wPaper;
    MoveL Offs(pOrigin,101.0,13.5,0.0),vDraw,z1,tPen\WObj:=wPaper;
    MoveL Offs(pOrigin,100.8,13.7,0.0),vDraw,z1,tPen\WObj:=wPaper;
    MoveL Offs(pOrigin,101.0,13.9,0.0),vDraw,z1,tPen\WObj:=wPaper;
    MoveL Offs(pOrigin,102.1,13.9,0.0),vDraw,z1,tPen\WObj:=wPaper;
    MoveL Offs(pOrigin,102.3,13.7,0.0),vDraw,fine,tPen\WObj:=wPaper;
    MoveL Offs(pOrigin,102.3,13.7,15.0),vApproach,z5,tPen\WObj:=wPaper;
    MoveL Offs(pOrigin,100.4,13.9,15.0),vTravel,z5,tPen\WObj:=wPaper;
    MoveL Offs(pOrigin,100.4,13.9,0.0),vApproach,fine,tPen\WObj:=wPaper;
    MoveL Offs(pOrigin,100.3,13.7,0.0),vDraw,z1,tPen\WObj:=wPaper;
    MoveL Offs(pOrigin,99.3,13.7,0.0),vDraw,z1,tPen\WObj:=wPaper;
    MoveL Offs(pOrigin,99.1,13.9,0.0),vDraw,z1,tPen\WObj:=wPaper;
    MoveL Offs(pOrigin,99.3,14.1,0.0),vDraw,z1,tPen\WObj:=wPaper;
    MoveL Offs(pOrigin,100.3,14.1,0.0),vDraw,z1,tPen\WObj:=wPaper;
    MoveL Offs(pOrigin,100.4,13.9,0.0),vDraw,fine,tPen\WObj:=wPaper;
    MoveL Offs(pOrigin,100.4,13.9,15.0),vApproach,z5,tPen\WObj:=wPaper;
    MoveL Offs(pOrigin,100.1,19.9,15.0),vTravel,z5,tPen\WObj:=wPaper;
    MoveL Offs(pOrigin,100.1,19.9,0.0),vApproach,fine,tPen\WObj:=wPaper;
    MoveL Offs(pOrigin,99.9,20.1,0.0),vDraw,z1,tPen\WObj:=wPaper;
    MoveL Offs(pOrigin,99.9,20.5,0.0),vDraw,z1,tPen\WObj:=wPaper;
    MoveL Offs(pOrigin,97.6,20.5,0.0),vDraw,z1,tPen\WObj:=wPaper;
    MoveL Offs(pOrigin,97.4,20.7,0.0),vDraw,z1,tPen\WObj:=wPaper;
    MoveL Offs(pOrigin,97.6,20.9,0.0),vDraw,z1,tPen\WObj:=wPaper;
    MoveL Offs(pOrigin,100.4,20.9,0.0),vDraw,z1,tPen\WObj:=wPaper;
    MoveL Offs(pOrigin,100.6,21.1,0.0),vDraw,z1,tPen\WObj:=wPaper;
    MoveL Offs(pOrigin,100.8,21.1,0.0),vDraw,z1,tPen\WObj:=wPaper;
    MoveL Offs(pOrigin,101.0,20.9,0.0),vDraw,z1,tPen\WObj:=wPaper;
    MoveL Offs(pOrigin,101.0,20.7,0.0),vDraw,z1,tPen\WObj:=wPaper;
    MoveL Offs(pOrigin,100.4,20.1,0.0),vDraw,z1,tPen\WObj:=wPaper;
    MoveL Offs(pOrigin,100.3,20.1,0.0),vDraw,z1,tPen\WObj:=wPaper;
    MoveL Offs(pOrigin,100.1,19.9,0.0),vDraw,fine,tPen\WObj:=wPaper;
    MoveL Offs(pOrigin,100.1,19.9,15.0),vApproach,z5,tPen\WObj:=wPaper;
    MoveL Offs(pOrigin,100.1,21.2,15.0),vTravel,z5,tPen\WObj:=wPaper;
    MoveL Offs(pOrigin,100.1,21.2,0.0),vApproach,fine,tPen\WObj:=wPaper;
    MoveL Offs(pOrigin,97.2,21.2,0.0),vDraw,z1,tPen\WObj:=wPaper;
    MoveL Offs(pOrigin,97.0,21.4,0.0),vDraw,z1,tPen\WObj:=wPaper;
    MoveL Offs(pOrigin,96.3,21.4,0.0),vDraw,z1,tPen\WObj:=wPaper;
    MoveL Offs(pOrigin,95.7,21.8,0.0),vDraw,z1,tPen\WObj:=wPaper;
    MoveL Offs(pOrigin,95.7,22.0,0.0),vDraw,z1,tPen\WObj:=wPaper;
    MoveL Offs(pOrigin,96.1,22.4,0.0),vDraw,z1,tPen\WObj:=wPaper;
    MoveL Offs(pOrigin,96.1,24.5,0.0),vDraw,z1,tPen\WObj:=wPaper;
    MoveL Offs(pOrigin,95.7,24.8,0.0),vDraw,z1,tPen\WObj:=wPaper;
    MoveL Offs(pOrigin,95.7,25.4,0.0),vDraw,z1,tPen\WObj:=wPaper;
    MoveL Offs(pOrigin,95.9,25.6,0.0),vDraw,z1,tPen\WObj:=wPaper;
    MoveL Offs(pOrigin,96.5,25.6,0.0),vDraw,z1,tPen\WObj:=wPaper;
    MoveL Offs(pOrigin,96.7,25.4,0.0),vDraw,z1,tPen\WObj:=wPaper;
    MoveL Offs(pOrigin,97.0,25.4,0.0),vDraw,z1,tPen\WObj:=wPaper;
    MoveL Offs(pOrigin,97.2,25.2,0.0),vDraw,z1,tPen\WObj:=wPaper;
    MoveL Offs(pOrigin,97.6,25.2,0.0),vDraw,z1,tPen\WObj:=wPaper;
    MoveL Offs(pOrigin,97.8,25.0,0.0),vDraw,z1,tPen\WObj:=wPaper;
    MoveL Offs(pOrigin,98.4,25.0,0.0),vDraw,z1,tPen\WObj:=wPaper;
    MoveL Offs(pOrigin,98.6,24.8,0.0),vDraw,z1,tPen\WObj:=wPaper;
    MoveL Offs(pOrigin,98.9,24.8,0.0),vDraw,z1,tPen\WObj:=wPaper;
    MoveL Offs(pOrigin,99.1,24.6,0.0),vDraw,z1,tPen\WObj:=wPaper;
    MoveL Offs(pOrigin,99.7,24.6,0.0),vDraw,z1,tPen\WObj:=wPaper;
    MoveL Offs(pOrigin,99.9,24.5,0.0),vDraw,z1,tPen\WObj:=wPaper;
    MoveL Offs(pOrigin,100.3,24.5,0.0),vDraw,z1,tPen\WObj:=wPaper;
    MoveL Offs(pOrigin,100.4,24.3,0.0),vDraw,z1,tPen\WObj:=wPaper;
    MoveL Offs(pOrigin,101.0,24.3,0.0),vDraw,z1,tPen\WObj:=wPaper;
    MoveL Offs(pOrigin,101.2,24.1,0.0),vDraw,z1,tPen\WObj:=wPaper;
    MoveL Offs(pOrigin,101.6,24.1,0.0),vDraw,z1,tPen\WObj:=wPaper;
    MoveL Offs(pOrigin,101.8,23.9,0.0),vDraw,z1,tPen\WObj:=wPaper;
    MoveL Offs(pOrigin,102.3,23.9,0.0),vDraw,z1,tPen\WObj:=wPaper;
    MoveL Offs(pOrigin,102.5,23.7,0.0),vDraw,z1,tPen\WObj:=wPaper;
    MoveL Offs(pOrigin,103.1,23.7,0.0),vDraw,z1,tPen\WObj:=wPaper;
    MoveL Offs(pOrigin,103.7,23.3,0.0),vDraw,z1,tPen\WObj:=wPaper;
    MoveL Offs(pOrigin,102.7,22.4,0.0),vDraw,z1,tPen\WObj:=wPaper;
    MoveL Offs(pOrigin,102.5,22.4,0.0),vDraw,z1,tPen\WObj:=wPaper;
    MoveL Offs(pOrigin,102.1,22.0,0.0),vDraw,z1,tPen\WObj:=wPaper;
    MoveL Offs(pOrigin,102.0,22.0,0.0),vDraw,z1,tPen\WObj:=wPaper;
    MoveL Offs(pOrigin,101.4,21.6,0.0),vDraw,z1,tPen\WObj:=wPaper;
    MoveL Offs(pOrigin,101.0,21.6,0.0),vDraw,z1,tPen\WObj:=wPaper;
    MoveL Offs(pOrigin,100.8,21.4,0.0),vDraw,z1,tPen\WObj:=wPaper;
    MoveL Offs(pOrigin,100.3,21.4,0.0),vDraw,z1,tPen\WObj:=wPaper;
    MoveL Offs(pOrigin,100.1,21.2,0.0),vDraw,fine,tPen\WObj:=wPaper;
    MoveL Offs(pOrigin,100.1,21.2,15.0),vApproach,z5,tPen\WObj:=wPaper;
    MoveL Offs(pOrigin,98.9,21.6,15.0),vTravel,z5,tPen\WObj:=wPaper;
  ENDPROC

  PROC Part105()
    MoveL Offs(pOrigin,98.9,21.6,0.0),vApproach,fine,tPen\WObj:=wPaper;
    MoveL Offs(pOrigin,98.9,22.0,0.0),vDraw,z1,tPen\WObj:=wPaper;
    MoveL Offs(pOrigin,99.3,22.4,0.0),vDraw,z1,tPen\WObj:=wPaper;
    MoveL Offs(pOrigin,99.7,22.4,0.0),vDraw,z1,tPen\WObj:=wPaper;
    MoveL Offs(pOrigin,99.7,22.6,0.0),vDraw,z1,tPen\WObj:=wPaper;
    MoveL Offs(pOrigin,99.9,22.8,0.0),vDraw,z1,tPen\WObj:=wPaper;
    MoveL Offs(pOrigin,99.9,23.1,0.0),vDraw,z1,tPen\WObj:=wPaper;
    MoveL Offs(pOrigin,99.7,23.1,0.0),vDraw,z1,tPen\WObj:=wPaper;
    MoveL Offs(pOrigin,99.5,23.3,0.0),vDraw,z1,tPen\WObj:=wPaper;
    MoveL Offs(pOrigin,99.5,23.5,0.0),vDraw,z1,tPen\WObj:=wPaper;
    MoveL Offs(pOrigin,99.3,23.7,0.0),vDraw,z1,tPen\WObj:=wPaper;
    MoveL Offs(pOrigin,99.3,24.1,0.0),vDraw,z1,tPen\WObj:=wPaper;
    MoveL Offs(pOrigin,98.7,24.1,0.0),vDraw,z1,tPen\WObj:=wPaper;
    MoveL Offs(pOrigin,98.7,23.9,0.0),vDraw,z1,tPen\WObj:=wPaper;
    MoveL Offs(pOrigin,98.4,23.3,0.0),vDraw,z1,tPen\WObj:=wPaper;
    MoveL Offs(pOrigin,98.4,22.9,0.0),vDraw,z1,tPen\WObj:=wPaper;
    MoveL Offs(pOrigin,98.2,22.8,0.0),vDraw,z1,tPen\WObj:=wPaper;
    MoveL Offs(pOrigin,98.2,21.6,0.0),vDraw,z1,tPen\WObj:=wPaper;
    MoveL Offs(pOrigin,98.9,21.6,0.0),vDraw,fine,tPen\WObj:=wPaper;
    MoveL Offs(pOrigin,98.9,21.6,15.0),vApproach,z5,tPen\WObj:=wPaper;
    MoveL Offs(pOrigin,95.0,22.9,15.0),vTravel,z5,tPen\WObj:=wPaper;
    MoveL Offs(pOrigin,95.0,22.9,0.0),vApproach,fine,tPen\WObj:=wPaper;
    MoveL Offs(pOrigin,94.4,22.4,0.0),vDraw,z1,tPen\WObj:=wPaper;
    MoveL Offs(pOrigin,94.2,22.4,0.0),vDraw,z1,tPen\WObj:=wPaper;
    MoveL Offs(pOrigin,94.2,22.2,0.0),vDraw,z1,tPen\WObj:=wPaper;
    MoveL Offs(pOrigin,94.0,22.0,0.0),vDraw,z1,tPen\WObj:=wPaper;
    MoveL Offs(pOrigin,93.8,22.2,0.0),vDraw,z1,tPen\WObj:=wPaper;
    MoveL Offs(pOrigin,93.6,22.2,0.0),vDraw,z1,tPen\WObj:=wPaper;
    MoveL Offs(pOrigin,93.1,22.8,0.0),vDraw,z1,tPen\WObj:=wPaper;
    MoveL Offs(pOrigin,93.1,22.9,0.0),vDraw,z1,tPen\WObj:=wPaper;
    MoveL Offs(pOrigin,92.9,23.1,0.0),vDraw,z1,tPen\WObj:=wPaper;
    MoveL Offs(pOrigin,92.9,23.5,0.0),vDraw,z1,tPen\WObj:=wPaper;
    MoveL Offs(pOrigin,93.6,24.3,0.0),vDraw,z1,tPen\WObj:=wPaper;
    MoveL Offs(pOrigin,94.0,24.3,0.0),vDraw,z1,tPen\WObj:=wPaper;
    MoveL Offs(pOrigin,94.2,24.1,0.0),vDraw,z1,tPen\WObj:=wPaper;
    MoveL Offs(pOrigin,94.8,24.1,0.0),vDraw,z1,tPen\WObj:=wPaper;
    MoveL Offs(pOrigin,95.2,23.5,0.0),vDraw,z1,tPen\WObj:=wPaper;
    MoveL Offs(pOrigin,95.0,22.9,0.0),vDraw,fine,tPen\WObj:=wPaper;
    MoveL Offs(pOrigin,95.0,22.9,15.0),vApproach,z5,tPen\WObj:=wPaper;
    MoveL Offs(pOrigin,94.8,18.6,15.0),vTravel,z5,tPen\WObj:=wPaper;
    MoveL Offs(pOrigin,94.8,18.6,0.0),vApproach,fine,tPen\WObj:=wPaper;
    MoveL Offs(pOrigin,95.0,18.4,0.0),vDraw,z1,tPen\WObj:=wPaper;
    MoveL Offs(pOrigin,94.8,18.2,0.0),vDraw,z1,tPen\WObj:=wPaper;
    MoveL Offs(pOrigin,92.3,18.2,0.0),vDraw,z1,tPen\WObj:=wPaper;
    MoveL Offs(pOrigin,92.1,18.4,0.0),vDraw,z1,tPen\WObj:=wPaper;
    MoveL Offs(pOrigin,92.3,18.6,0.0),vDraw,z1,tPen\WObj:=wPaper;
    MoveL Offs(pOrigin,94.8,18.6,0.0),vDraw,fine,tPen\WObj:=wPaper;
    MoveL Offs(pOrigin,94.8,18.6,15.0),vApproach,z5,tPen\WObj:=wPaper;
    MoveL Offs(pOrigin,90.6,18.6,15.0),vTravel,z5,tPen\WObj:=wPaper;
    MoveL Offs(pOrigin,90.6,18.6,0.0),vApproach,fine,tPen\WObj:=wPaper;
    MoveL Offs(pOrigin,90.4,18.4,0.0),vDraw,z1,tPen\WObj:=wPaper;
    MoveL Offs(pOrigin,88.4,18.4,0.0),vDraw,z1,tPen\WObj:=wPaper;
    MoveL Offs(pOrigin,88.2,18.6,0.0),vDraw,z1,tPen\WObj:=wPaper;
    MoveL Offs(pOrigin,88.4,18.8,0.0),vDraw,z1,tPen\WObj:=wPaper;
    MoveL Offs(pOrigin,90.4,18.8,0.0),vDraw,z1,tPen\WObj:=wPaper;
    MoveL Offs(pOrigin,90.6,18.6,0.0),vDraw,fine,tPen\WObj:=wPaper;
    MoveL Offs(pOrigin,90.6,18.6,15.0),vApproach,z5,tPen\WObj:=wPaper;
    MoveL Offs(pOrigin,87.8,19.5,15.0),vTravel,z5,tPen\WObj:=wPaper;
    MoveL Offs(pOrigin,87.8,19.5,0.0),vApproach,fine,tPen\WObj:=wPaper;
    MoveL Offs(pOrigin,87.8,19.9,0.0),vDraw,z1,tPen\WObj:=wPaper;
    MoveL Offs(pOrigin,87.4,19.9,0.0),vDraw,z1,tPen\WObj:=wPaper;
    MoveL Offs(pOrigin,87.2,20.1,0.0),vDraw,z1,tPen\WObj:=wPaper;
    MoveL Offs(pOrigin,86.3,20.3,0.0),vDraw,z1,tPen\WObj:=wPaper;
    MoveL Offs(pOrigin,86.3,19.5,0.0),vDraw,z1,tPen\WObj:=wPaper;
    MoveL Offs(pOrigin,86.5,19.4,0.0),vDraw,z1,tPen\WObj:=wPaper;
    MoveL Offs(pOrigin,87.0,19.4,0.0),vDraw,z1,tPen\WObj:=wPaper;
    MoveL Offs(pOrigin,87.2,19.5,0.0),vDraw,z1,tPen\WObj:=wPaper;
    MoveL Offs(pOrigin,87.8,19.5,0.0),vDraw,fine,tPen\WObj:=wPaper;
    MoveL Offs(pOrigin,87.8,19.5,15.0),vApproach,z5,tPen\WObj:=wPaper;
    MoveL Offs(pOrigin,85.5,18.6,15.0),vTravel,z5,tPen\WObj:=wPaper;
    MoveL Offs(pOrigin,85.5,18.6,0.0),vApproach,fine,tPen\WObj:=wPaper;
    MoveL Offs(pOrigin,85.3,18.4,0.0),vDraw,z1,tPen\WObj:=wPaper;
    MoveL Offs(pOrigin,84.4,18.4,0.0),vDraw,z1,tPen\WObj:=wPaper;
    MoveL Offs(pOrigin,84.2,18.6,0.0),vDraw,z1,tPen\WObj:=wPaper;
    MoveL Offs(pOrigin,84.4,18.8,0.0),vDraw,z1,tPen\WObj:=wPaper;
    MoveL Offs(pOrigin,85.3,18.8,0.0),vDraw,z1,tPen\WObj:=wPaper;
    MoveL Offs(pOrigin,85.5,18.6,0.0),vDraw,fine,tPen\WObj:=wPaper;
    MoveL Offs(pOrigin,85.5,18.6,15.0),vApproach,z5,tPen\WObj:=wPaper;
    MoveL Offs(pOrigin,81.6,22.8,15.0),vTravel,z5,tPen\WObj:=wPaper;
    MoveL Offs(pOrigin,81.6,22.8,0.0),vApproach,fine,tPen\WObj:=wPaper;
    MoveL Offs(pOrigin,81.6,23.1,0.0),vDraw,z1,tPen\WObj:=wPaper;
    MoveL Offs(pOrigin,81.4,23.3,0.0),vDraw,z1,tPen\WObj:=wPaper;
    MoveL Offs(pOrigin,81.4,24.3,0.0),vDraw,z1,tPen\WObj:=wPaper;
    MoveL Offs(pOrigin,81.2,24.5,0.0),vDraw,z1,tPen\WObj:=wPaper;
    MoveL Offs(pOrigin,81.2,25.2,0.0),vDraw,z1,tPen\WObj:=wPaper;
    MoveL Offs(pOrigin,81.4,25.4,0.0),vDraw,z1,tPen\WObj:=wPaper;
    MoveL Offs(pOrigin,81.4,26.3,0.0),vDraw,z1,tPen\WObj:=wPaper;
    MoveL Offs(pOrigin,81.6,26.5,0.0),vDraw,z1,tPen\WObj:=wPaper;
    MoveL Offs(pOrigin,81.6,27.1,0.0),vDraw,z1,tPen\WObj:=wPaper;
    MoveL Offs(pOrigin,81.7,27.3,0.0),vDraw,z1,tPen\WObj:=wPaper;
    MoveL Offs(pOrigin,81.7,27.7,0.0),vDraw,z1,tPen\WObj:=wPaper;
    MoveL Offs(pOrigin,81.9,27.9,0.0),vDraw,z1,tPen\WObj:=wPaper;
    MoveL Offs(pOrigin,81.9,28.4,0.0),vDraw,z1,tPen\WObj:=wPaper;
    MoveL Offs(pOrigin,81.7,28.6,0.0),vDraw,z1,tPen\WObj:=wPaper;
    MoveL Offs(pOrigin,81.7,29.0,0.0),vDraw,z1,tPen\WObj:=wPaper;
    MoveL Offs(pOrigin,81.4,29.0,0.0),vDraw,z1,tPen\WObj:=wPaper;
    MoveL Offs(pOrigin,81.2,28.8,0.0),vDraw,z1,tPen\WObj:=wPaper;
    MoveL Offs(pOrigin,81.2,28.6,0.0),vDraw,z1,tPen\WObj:=wPaper;
    MoveL Offs(pOrigin,80.8,28.0,0.0),vDraw,z1,tPen\WObj:=wPaper;
    MoveL Offs(pOrigin,80.8,27.7,0.0),vDraw,z1,tPen\WObj:=wPaper;
    MoveL Offs(pOrigin,80.6,27.5,0.0),vDraw,z1,tPen\WObj:=wPaper;
    MoveL Offs(pOrigin,80.6,26.7,0.0),vDraw,z1,tPen\WObj:=wPaper;
    MoveL Offs(pOrigin,80.4,26.5,0.0),vDraw,z1,tPen\WObj:=wPaper;
    MoveL Offs(pOrigin,80.4,23.3,0.0),vDraw,z1,tPen\WObj:=wPaper;
    MoveL Offs(pOrigin,80.6,23.1,0.0),vDraw,z1,tPen\WObj:=wPaper;
    MoveL Offs(pOrigin,80.6,22.8,0.0),vDraw,z1,tPen\WObj:=wPaper;
    MoveL Offs(pOrigin,80.8,22.6,0.0),vDraw,z1,tPen\WObj:=wPaper;
    MoveL Offs(pOrigin,80.8,22.4,0.0),vDraw,z1,tPen\WObj:=wPaper;
    MoveL Offs(pOrigin,81.2,22.4,0.0),vDraw,z1,tPen\WObj:=wPaper;
    MoveL Offs(pOrigin,81.2,22.6,0.0),vDraw,z1,tPen\WObj:=wPaper;
    MoveL Offs(pOrigin,81.4,22.8,0.0),vDraw,z1,tPen\WObj:=wPaper;
    MoveL Offs(pOrigin,81.6,22.8,0.0),vDraw,fine,tPen\WObj:=wPaper;
    MoveL Offs(pOrigin,81.6,22.8,15.0),vApproach,z5,tPen\WObj:=wPaper;
    MoveL Offs(pOrigin,79.7,21.4,15.0),vTravel,z5,tPen\WObj:=wPaper;
    MoveL Offs(pOrigin,79.7,21.4,0.0),vApproach,fine,tPen\WObj:=wPaper;
    MoveL Offs(pOrigin,79.7,21.2,0.0),vDraw,z1,tPen\WObj:=wPaper;
    MoveL Offs(pOrigin,79.5,21.1,0.0),vDraw,z1,tPen\WObj:=wPaper;
    MoveL Offs(pOrigin,79.1,21.4,0.0),vDraw,z1,tPen\WObj:=wPaper;
    MoveL Offs(pOrigin,78.9,21.4,0.0),vDraw,z1,tPen\WObj:=wPaper;
    MoveL Offs(pOrigin,78.3,21.8,0.0),vDraw,z1,tPen\WObj:=wPaper;
  ENDPROC

  PROC Part106()
    MoveL Offs(pOrigin,78.5,22.0,0.0),vDraw,z1,tPen\WObj:=wPaper;
    MoveL Offs(pOrigin,78.9,22.0,0.0),vDraw,z1,tPen\WObj:=wPaper;
    MoveL Offs(pOrigin,79.1,22.2,0.0),vDraw,z1,tPen\WObj:=wPaper;
    MoveL Offs(pOrigin,79.7,21.4,0.0),vDraw,fine,tPen\WObj:=wPaper;
    MoveL Offs(pOrigin,79.7,21.4,15.0),vApproach,z5,tPen\WObj:=wPaper;
    MoveL Offs(pOrigin,78.3,21.1,15.0),vTravel,z5,tPen\WObj:=wPaper;
    MoveL Offs(pOrigin,78.3,21.1,0.0),vApproach,fine,tPen\WObj:=wPaper;
    MoveL Offs(pOrigin,78.2,20.9,0.0),vDraw,z1,tPen\WObj:=wPaper;
    MoveL Offs(pOrigin,76.5,20.9,0.0),vDraw,z1,tPen\WObj:=wPaper;
    MoveL Offs(pOrigin,76.3,21.1,0.0),vDraw,z1,tPen\WObj:=wPaper;
    MoveL Offs(pOrigin,76.5,21.2,0.0),vDraw,z1,tPen\WObj:=wPaper;
    MoveL Offs(pOrigin,76.8,21.2,0.0),vDraw,z1,tPen\WObj:=wPaper;
    MoveL Offs(pOrigin,76.8,21.8,0.0),vDraw,z1,tPen\WObj:=wPaper;
    MoveL Offs(pOrigin,77.0,22.0,0.0),vDraw,z1,tPen\WObj:=wPaper;
    MoveL Offs(pOrigin,77.4,21.6,0.0),vDraw,z1,tPen\WObj:=wPaper;
    MoveL Offs(pOrigin,78.0,21.4,0.0),vDraw,z1,tPen\WObj:=wPaper;
    MoveL Offs(pOrigin,78.3,21.1,0.0),vDraw,fine,tPen\WObj:=wPaper;
    MoveL Offs(pOrigin,78.3,21.1,15.0),vApproach,z5,tPen\WObj:=wPaper;
    MoveL Offs(pOrigin,76.5,22.2,15.0),vTravel,z5,tPen\WObj:=wPaper;
    MoveL Offs(pOrigin,76.5,22.2,0.0),vApproach,fine,tPen\WObj:=wPaper;
    MoveL Offs(pOrigin,76.3,22.0,0.0),vDraw,z1,tPen\WObj:=wPaper;
    MoveL Offs(pOrigin,75.1,22.0,0.0),vDraw,z1,tPen\WObj:=wPaper;
    MoveL Offs(pOrigin,74.9,22.2,0.0),vDraw,z1,tPen\WObj:=wPaper;
    MoveL Offs(pOrigin,74.9,22.6,0.0),vDraw,z1,tPen\WObj:=wPaper;
    MoveL Offs(pOrigin,75.1,22.8,0.0),vDraw,z1,tPen\WObj:=wPaper;
    MoveL Offs(pOrigin,75.5,22.8,0.0),vDraw,z1,tPen\WObj:=wPaper;
    MoveL Offs(pOrigin,76.5,22.2,0.0),vDraw,fine,tPen\WObj:=wPaper;
    MoveL Offs(pOrigin,76.5,22.2,15.0),vApproach,z5,tPen\WObj:=wPaper;
    MoveL Offs(pOrigin,74.6,20.7,15.0),vTravel,z5,tPen\WObj:=wPaper;
    MoveL Offs(pOrigin,74.6,20.7,0.0),vApproach,fine,tPen\WObj:=wPaper;
    MoveL Offs(pOrigin,74.4,20.5,0.0),vDraw,z1,tPen\WObj:=wPaper;
    MoveL Offs(pOrigin,73.1,20.5,0.0),vDraw,z1,tPen\WObj:=wPaper;
    MoveL Offs(pOrigin,72.9,20.7,0.0),vDraw,z1,tPen\WObj:=wPaper;
    MoveL Offs(pOrigin,73.1,20.9,0.0),vDraw,z1,tPen\WObj:=wPaper;
    MoveL Offs(pOrigin,74.4,20.9,0.0),vDraw,z1,tPen\WObj:=wPaper;
    MoveL Offs(pOrigin,74.6,20.7,0.0),vDraw,fine,tPen\WObj:=wPaper;
    MoveL Offs(pOrigin,74.6,20.7,15.0),vApproach,z5,tPen\WObj:=wPaper;
    MoveL Offs(pOrigin,72.7,20.9,15.0),vTravel,z5,tPen\WObj:=wPaper;
    MoveL Offs(pOrigin,72.7,20.9,0.0),vApproach,fine,tPen\WObj:=wPaper;
    MoveL Offs(pOrigin,72.5,20.7,0.0),vDraw,z1,tPen\WObj:=wPaper;
    MoveL Offs(pOrigin,71.0,20.7,0.0),vDraw,z1,tPen\WObj:=wPaper;
    MoveL Offs(pOrigin,70.8,20.9,0.0),vDraw,z1,tPen\WObj:=wPaper;
    MoveL Offs(pOrigin,71.0,21.1,0.0),vDraw,z1,tPen\WObj:=wPaper;
    MoveL Offs(pOrigin,71.4,21.1,0.0),vDraw,z1,tPen\WObj:=wPaper;
    MoveL Offs(pOrigin,71.5,21.2,0.0),vDraw,z1,tPen\WObj:=wPaper;
    MoveL Offs(pOrigin,71.9,21.2,0.0),vDraw,z1,tPen\WObj:=wPaper;
    MoveL Offs(pOrigin,72.1,21.1,0.0),vDraw,z1,tPen\WObj:=wPaper;
    MoveL Offs(pOrigin,72.5,21.1,0.0),vDraw,z1,tPen\WObj:=wPaper;
    MoveL Offs(pOrigin,72.7,20.9,0.0),vDraw,fine,tPen\WObj:=wPaper;
    MoveL Offs(pOrigin,72.7,20.9,15.0),vApproach,z5,tPen\WObj:=wPaper;
    MoveL Offs(pOrigin,98.9,26.9,15.0),vTravel,z5,tPen\WObj:=wPaper;
    MoveL Offs(pOrigin,98.9,26.9,0.0),vApproach,fine,tPen\WObj:=wPaper;
    MoveL Offs(pOrigin,99.3,26.9,0.0),vDraw,z1,tPen\WObj:=wPaper;
    MoveL Offs(pOrigin,99.9,26.3,0.0),vDraw,z1,tPen\WObj:=wPaper;
    MoveL Offs(pOrigin,100.8,26.3,0.0),vDraw,z1,tPen\WObj:=wPaper;
    MoveL Offs(pOrigin,101.4,26.9,0.0),vDraw,z1,tPen\WObj:=wPaper;
    MoveL Offs(pOrigin,101.4,27.1,0.0),vDraw,z1,tPen\WObj:=wPaper;
    MoveL Offs(pOrigin,101.6,27.3,0.0),vDraw,z1,tPen\WObj:=wPaper;
    MoveL Offs(pOrigin,101.6,27.7,0.0),vDraw,z1,tPen\WObj:=wPaper;
    MoveL Offs(pOrigin,101.8,27.9,0.0),vDraw,z1,tPen\WObj:=wPaper;
    MoveL Offs(pOrigin,101.8,29.4,0.0),vDraw,z1,tPen\WObj:=wPaper;
    MoveL Offs(pOrigin,100.8,29.2,0.0),vDraw,z1,tPen\WObj:=wPaper;
    MoveL Offs(pOrigin,100.6,29.4,0.0),vDraw,z1,tPen\WObj:=wPaper;
    MoveL Offs(pOrigin,100.6,29.7,0.0),vDraw,z1,tPen\WObj:=wPaper;
    MoveL Offs(pOrigin,100.4,29.9,0.0),vDraw,z1,tPen\WObj:=wPaper;
    MoveL Offs(pOrigin,100.4,30.1,0.0),vDraw,z1,tPen\WObj:=wPaper;
    MoveL Offs(pOrigin,99.9,30.1,0.0),vDraw,z1,tPen\WObj:=wPaper;
    MoveL Offs(pOrigin,99.1,29.2,0.0),vDraw,z1,tPen\WObj:=wPaper;
    MoveL Offs(pOrigin,99.1,28.8,0.0),vDraw,z1,tPen\WObj:=wPaper;
    MoveL Offs(pOrigin,98.9,28.6,0.0),vDraw,z1,tPen\WObj:=wPaper;
    MoveL Offs(pOrigin,98.9,26.9,0.0),vDraw,fine,tPen\WObj:=wPaper;
    MoveL Offs(pOrigin,98.9,26.9,15.0),vApproach,z5,tPen\WObj:=wPaper;
    MoveL Offs(pOrigin,104.2,23.9,15.0),vTravel,z5,tPen\WObj:=wPaper;
    MoveL Offs(pOrigin,104.2,23.9,0.0),vApproach,fine,tPen\WObj:=wPaper;
    MoveL Offs(pOrigin,104.4,24.1,0.0),vDraw,z1,tPen\WObj:=wPaper;
    MoveL Offs(pOrigin,104.6,24.1,0.0),vDraw,z1,tPen\WObj:=wPaper;
    MoveL Offs(pOrigin,104.8,23.9,0.0),vDraw,z1,tPen\WObj:=wPaper;
    MoveL Offs(pOrigin,105.9,23.9,0.0),vDraw,z1,tPen\WObj:=wPaper;
    MoveL Offs(pOrigin,106.1,24.1,0.0),vDraw,z1,tPen\WObj:=wPaper;
    MoveL Offs(pOrigin,106.7,24.1,0.0),vDraw,z1,tPen\WObj:=wPaper;
    MoveL Offs(pOrigin,106.9,23.9,0.0),vDraw,z1,tPen\WObj:=wPaper;
    MoveL Offs(pOrigin,106.9,23.5,0.0),vDraw,z1,tPen\WObj:=wPaper;
    MoveL Offs(pOrigin,108.8,23.5,0.0),vDraw,z1,tPen\WObj:=wPaper;
    MoveL Offs(pOrigin,109.1,24.1,0.0),vDraw,z1,tPen\WObj:=wPaper;
    MoveL Offs(pOrigin,109.3,23.9,0.0),vDraw,z1,tPen\WObj:=wPaper;
    MoveL Offs(pOrigin,109.3,23.3,0.0),vDraw,z1,tPen\WObj:=wPaper;
    MoveL Offs(pOrigin,110.5,23.3,0.0),vDraw,z1,tPen\WObj:=wPaper;
    MoveL Offs(pOrigin,110.6,23.1,0.0),vDraw,z1,tPen\WObj:=wPaper;
    MoveL Offs(pOrigin,110.5,22.9,0.0),vDraw,z1,tPen\WObj:=wPaper;
    MoveL Offs(pOrigin,108.8,22.9,0.0),vDraw,z1,tPen\WObj:=wPaper;
    MoveL Offs(pOrigin,108.6,23.1,0.0),vDraw,z1,tPen\WObj:=wPaper;
    MoveL Offs(pOrigin,106.5,23.1,0.0),vDraw,z1,tPen\WObj:=wPaper;
    MoveL Offs(pOrigin,106.3,23.3,0.0),vDraw,z1,tPen\WObj:=wPaper;
    MoveL Offs(pOrigin,104.8,23.3,0.0),vDraw,z1,tPen\WObj:=wPaper;
    MoveL Offs(pOrigin,104.4,22.9,0.0),vDraw,z1,tPen\WObj:=wPaper;
    MoveL Offs(pOrigin,104.2,23.1,0.0),vDraw,z1,tPen\WObj:=wPaper;
    MoveL Offs(pOrigin,104.2,23.9,0.0),vDraw,fine,tPen\WObj:=wPaper;
    MoveL Offs(pOrigin,104.2,23.9,15.0),vApproach,z5,tPen\WObj:=wPaper;
    MoveL Offs(pOrigin,106.9,25.6,15.0),vTravel,z5,tPen\WObj:=wPaper;
    MoveL Offs(pOrigin,106.9,25.6,0.0),vApproach,fine,tPen\WObj:=wPaper;
    MoveL Offs(pOrigin,106.9,26.3,0.0),vDraw,z1,tPen\WObj:=wPaper;
    MoveL Offs(pOrigin,107.1,26.5,0.0),vDraw,z1,tPen\WObj:=wPaper;
    MoveL Offs(pOrigin,107.2,26.3,0.0),vDraw,z1,tPen\WObj:=wPaper;
    MoveL Offs(pOrigin,107.2,25.6,0.0),vDraw,z1,tPen\WObj:=wPaper;
    MoveL Offs(pOrigin,107.1,25.4,0.0),vDraw,z1,tPen\WObj:=wPaper;
    MoveL Offs(pOrigin,106.9,25.6,0.0),vDraw,fine,tPen\WObj:=wPaper;
    MoveL Offs(pOrigin,106.9,25.6,15.0),vApproach,z5,tPen\WObj:=wPaper;
    MoveL Offs(pOrigin,107.6,25.6,15.0),vTravel,z5,tPen\WObj:=wPaper;
    MoveL Offs(pOrigin,107.6,25.6,0.0),vApproach,fine,tPen\WObj:=wPaper;
    MoveL Offs(pOrigin,107.6,26.5,0.0),vDraw,z1,tPen\WObj:=wPaper;
    MoveL Offs(pOrigin,107.8,26.7,0.0),vDraw,z1,tPen\WObj:=wPaper;
    MoveL Offs(pOrigin,108.4,26.2,0.0),vDraw,z1,tPen\WObj:=wPaper;
    MoveL Offs(pOrigin,108.2,26.0,0.0),vDraw,z1,tPen\WObj:=wPaper;
    MoveL Offs(pOrigin,108.0,26.0,0.0),vDraw,z1,tPen\WObj:=wPaper;
    MoveL Offs(pOrigin,108.0,25.6,0.0),vDraw,z1,tPen\WObj:=wPaper;
    MoveL Offs(pOrigin,107.8,25.4,0.0),vDraw,z1,tPen\WObj:=wPaper;
    MoveL Offs(pOrigin,107.6,25.6,0.0),vDraw,fine,tPen\WObj:=wPaper;
    MoveL Offs(pOrigin,107.6,25.6,15.0),vApproach,z5,tPen\WObj:=wPaper;
    MoveL Offs(pOrigin,108.2,25.0,15.0),vTravel,z5,tPen\WObj:=wPaper;
    MoveL Offs(pOrigin,108.2,25.0,0.0),vApproach,fine,tPen\WObj:=wPaper;
  ENDPROC

  PROC Part107()
    MoveL Offs(pOrigin,108.4,25.2,0.0),vDraw,z1,tPen\WObj:=wPaper;
    MoveL Offs(pOrigin,108.6,25.2,0.0),vDraw,z1,tPen\WObj:=wPaper;
    MoveL Offs(pOrigin,108.8,25.0,0.0),vDraw,z1,tPen\WObj:=wPaper;
    MoveL Offs(pOrigin,108.8,24.6,0.0),vDraw,z1,tPen\WObj:=wPaper;
    MoveL Offs(pOrigin,108.6,24.5,0.0),vDraw,z1,tPen\WObj:=wPaper;
    MoveL Offs(pOrigin,108.6,24.3,0.0),vDraw,z1,tPen\WObj:=wPaper;
    MoveL Offs(pOrigin,108.2,23.9,0.0),vDraw,z1,tPen\WObj:=wPaper;
    MoveL Offs(pOrigin,108.0,23.9,0.0),vDraw,z1,tPen\WObj:=wPaper;
    MoveL Offs(pOrigin,107.8,24.1,0.0),vDraw,z1,tPen\WObj:=wPaper;
    MoveL Offs(pOrigin,108.2,24.6,0.0),vDraw,z1,tPen\WObj:=wPaper;
    MoveL Offs(pOrigin,108.2,25.0,0.0),vDraw,fine,tPen\WObj:=wPaper;
    MoveL Offs(pOrigin,108.2,25.0,15.0),vApproach,z5,tPen\WObj:=wPaper;
    MoveL Offs(pOrigin,108.9,26.5,15.0),vTravel,z5,tPen\WObj:=wPaper;
    MoveL Offs(pOrigin,108.9,26.5,0.0),vApproach,fine,tPen\WObj:=wPaper;
    MoveL Offs(pOrigin,108.2,27.3,0.0),vDraw,z1,tPen\WObj:=wPaper;
    MoveL Offs(pOrigin,108.2,27.5,0.0),vDraw,z1,tPen\WObj:=wPaper;
    MoveL Offs(pOrigin,108.4,27.7,0.0),vDraw,z1,tPen\WObj:=wPaper;
    MoveL Offs(pOrigin,108.8,27.3,0.0),vDraw,z1,tPen\WObj:=wPaper;
    MoveL Offs(pOrigin,108.9,27.3,0.0),vDraw,z1,tPen\WObj:=wPaper;
    MoveL Offs(pOrigin,109.9,26.3,0.0),vDraw,z1,tPen\WObj:=wPaper;
    MoveL Offs(pOrigin,110.5,26.3,0.0),vDraw,z1,tPen\WObj:=wPaper;
    MoveL Offs(pOrigin,111.0,25.6,0.0),vDraw,z1,tPen\WObj:=wPaper;
    MoveL Offs(pOrigin,110.8,25.4,0.0),vDraw,z1,tPen\WObj:=wPaper;
    MoveL Offs(pOrigin,110.3,25.6,0.0),vDraw,z1,tPen\WObj:=wPaper;
    MoveL Offs(pOrigin,109.1,26.5,0.0),vDraw,z1,tPen\WObj:=wPaper;
    MoveL Offs(pOrigin,108.9,26.5,0.0),vDraw,fine,tPen\WObj:=wPaper;
    MoveL Offs(pOrigin,108.9,26.5,15.0),vApproach,z5,tPen\WObj:=wPaper;
    MoveL Offs(pOrigin,110.1,27.9,15.0),vTravel,z5,tPen\WObj:=wPaper;
    MoveL Offs(pOrigin,110.1,27.9,0.0),vApproach,fine,tPen\WObj:=wPaper;
    MoveL Offs(pOrigin,110.3,28.0,0.0),vDraw,z1,tPen\WObj:=wPaper;
    MoveL Offs(pOrigin,110.8,28.0,0.0),vDraw,z1,tPen\WObj:=wPaper;
    MoveL Offs(pOrigin,111.0,27.9,0.0),vDraw,z1,tPen\WObj:=wPaper;
    MoveL Offs(pOrigin,111.0,27.1,0.0),vDraw,z1,tPen\WObj:=wPaper;
    MoveL Offs(pOrigin,110.8,26.9,0.0),vDraw,z1,tPen\WObj:=wPaper;
    MoveL Offs(pOrigin,110.6,27.1,0.0),vDraw,z1,tPen\WObj:=wPaper;
    MoveL Offs(pOrigin,110.6,27.3,0.0),vDraw,z1,tPen\WObj:=wPaper;
    MoveL Offs(pOrigin,110.1,27.9,0.0),vDraw,fine,tPen\WObj:=wPaper;
    MoveL Offs(pOrigin,110.1,27.9,15.0),vApproach,z5,tPen\WObj:=wPaper;
    MoveL Offs(pOrigin,111.4,27.7,15.0),vTravel,z5,tPen\WObj:=wPaper;
    MoveL Offs(pOrigin,111.4,27.7,0.0),vApproach,fine,tPen\WObj:=wPaper;
    MoveL Offs(pOrigin,111.6,27.9,0.0),vDraw,z1,tPen\WObj:=wPaper;
    MoveL Offs(pOrigin,111.6,28.2,0.0),vDraw,z1,tPen\WObj:=wPaper;
    MoveL Offs(pOrigin,111.8,28.4,0.0),vDraw,z1,tPen\WObj:=wPaper;
    MoveL Offs(pOrigin,111.8,28.8,0.0),vDraw,z1,tPen\WObj:=wPaper;
    MoveL Offs(pOrigin,112.0,29.0,0.0),vDraw,z1,tPen\WObj:=wPaper;
    MoveL Offs(pOrigin,112.0,29.4,0.0),vDraw,z1,tPen\WObj:=wPaper;
    MoveL Offs(pOrigin,112.2,29.6,0.0),vDraw,z1,tPen\WObj:=wPaper;
    MoveL Offs(pOrigin,112.2,29.9,0.0),vDraw,z1,tPen\WObj:=wPaper;
    MoveL Offs(pOrigin,112.3,30.1,0.0),vDraw,z1,tPen\WObj:=wPaper;
    MoveL Offs(pOrigin,112.3,30.5,0.0),vDraw,z1,tPen\WObj:=wPaper;
    MoveL Offs(pOrigin,112.5,30.7,0.0),vDraw,z1,tPen\WObj:=wPaper;
    MoveL Offs(pOrigin,112.5,31.3,0.0),vDraw,z1,tPen\WObj:=wPaper;
    MoveL Offs(pOrigin,112.7,31.4,0.0),vDraw,z1,tPen\WObj:=wPaper;
    MoveL Offs(pOrigin,112.7,31.8,0.0),vDraw,z1,tPen\WObj:=wPaper;
    MoveL Offs(pOrigin,112.9,32.0,0.0),vDraw,z1,tPen\WObj:=wPaper;
    MoveL Offs(pOrigin,112.9,32.4,0.0),vDraw,z1,tPen\WObj:=wPaper;
    MoveL Offs(pOrigin,113.1,32.6,0.0),vDraw,z1,tPen\WObj:=wPaper;
    MoveL Offs(pOrigin,113.1,33.1,0.0),vDraw,z1,tPen\WObj:=wPaper;
    MoveL Offs(pOrigin,113.3,33.3,0.0),vDraw,z1,tPen\WObj:=wPaper;
    MoveL Offs(pOrigin,113.3,33.9,0.0),vDraw,z1,tPen\WObj:=wPaper;
    MoveL Offs(pOrigin,113.7,34.3,0.0),vDraw,z1,tPen\WObj:=wPaper;
    MoveL Offs(pOrigin,114.2,33.5,0.0),vDraw,z1,tPen\WObj:=wPaper;
    MoveL Offs(pOrigin,114.2,33.3,0.0),vDraw,z1,tPen\WObj:=wPaper;
    MoveL Offs(pOrigin,114.8,32.8,0.0),vDraw,z1,tPen\WObj:=wPaper;
    MoveL Offs(pOrigin,114.8,32.6,0.0),vDraw,z1,tPen\WObj:=wPaper;
    MoveL Offs(pOrigin,115.2,32.2,0.0),vDraw,z1,tPen\WObj:=wPaper;
    MoveL Offs(pOrigin,115.2,32.0,0.0),vDraw,z1,tPen\WObj:=wPaper;
    MoveL Offs(pOrigin,115.6,31.6,0.0),vDraw,z1,tPen\WObj:=wPaper;
    MoveL Offs(pOrigin,115.6,31.4,0.0),vDraw,z1,tPen\WObj:=wPaper;
    MoveL Offs(pOrigin,115.9,31.1,0.0),vDraw,z1,tPen\WObj:=wPaper;
    MoveL Offs(pOrigin,115.9,30.9,0.0),vDraw,z1,tPen\WObj:=wPaper;
    MoveL Offs(pOrigin,116.3,30.5,0.0),vDraw,z1,tPen\WObj:=wPaper;
    MoveL Offs(pOrigin,116.5,29.9,0.0),vDraw,z1,tPen\WObj:=wPaper;
    MoveL Offs(pOrigin,117.6,28.4,0.0),vDraw,z1,tPen\WObj:=wPaper;
    MoveL Offs(pOrigin,117.6,28.2,0.0),vDraw,z1,tPen\WObj:=wPaper;
    MoveL Offs(pOrigin,118.2,27.5,0.0),vDraw,z1,tPen\WObj:=wPaper;
    MoveL Offs(pOrigin,118.2,27.3,0.0),vDraw,z1,tPen\WObj:=wPaper;
    MoveL Offs(pOrigin,118.8,27.3,0.0),vDraw,z1,tPen\WObj:=wPaper;
    MoveL Offs(pOrigin,118.8,27.7,0.0),vDraw,z1,tPen\WObj:=wPaper;
    MoveL Offs(pOrigin,118.6,27.9,0.0),vDraw,z1,tPen\WObj:=wPaper;
    MoveL Offs(pOrigin,118.8,28.0,0.0),vDraw,z1,tPen\WObj:=wPaper;
    MoveL Offs(pOrigin,119.0,28.0,0.0),vDraw,z1,tPen\WObj:=wPaper;
    MoveL Offs(pOrigin,119.1,27.9,0.0),vDraw,z1,tPen\WObj:=wPaper;
    MoveL Offs(pOrigin,119.1,26.9,0.0),vDraw,z1,tPen\WObj:=wPaper;
    MoveL Offs(pOrigin,119.0,26.7,0.0),vDraw,z1,tPen\WObj:=wPaper;
    MoveL Offs(pOrigin,119.0,24.1,0.0),vDraw,z1,tPen\WObj:=wPaper;
    MoveL Offs(pOrigin,118.8,23.9,0.0),vDraw,z1,tPen\WObj:=wPaper;
    MoveL Offs(pOrigin,118.8,23.3,0.0),vDraw,z1,tPen\WObj:=wPaper;
    MoveL Offs(pOrigin,118.6,23.1,0.0),vDraw,z1,tPen\WObj:=wPaper;
    MoveL Offs(pOrigin,116.3,23.1,0.0),vDraw,z1,tPen\WObj:=wPaper;
    MoveL Offs(pOrigin,116.1,23.3,0.0),vDraw,z1,tPen\WObj:=wPaper;
    MoveL Offs(pOrigin,114.2,23.3,0.0),vDraw,z1,tPen\WObj:=wPaper;
    MoveL Offs(pOrigin,113.7,23.9,0.0),vDraw,z1,tPen\WObj:=wPaper;
    MoveL Offs(pOrigin,113.3,24.8,0.0),vDraw,z1,tPen\WObj:=wPaper;
    MoveL Offs(pOrigin,112.9,25.2,0.0),vDraw,z1,tPen\WObj:=wPaper;
    MoveL Offs(pOrigin,112.9,25.4,0.0),vDraw,z1,tPen\WObj:=wPaper;
    MoveL Offs(pOrigin,112.5,25.8,0.0),vDraw,z1,tPen\WObj:=wPaper;
    MoveL Offs(pOrigin,112.5,26.0,0.0),vDraw,z1,tPen\WObj:=wPaper;
    MoveL Offs(pOrigin,111.4,27.3,0.0),vDraw,z1,tPen\WObj:=wPaper;
    MoveL Offs(pOrigin,111.4,27.7,0.0),vDraw,fine,tPen\WObj:=wPaper;
    MoveL Offs(pOrigin,111.4,27.7,15.0),vApproach,z5,tPen\WObj:=wPaper;
    MoveL Offs(pOrigin,108.8,29.4,15.0),vTravel,z5,tPen\WObj:=wPaper;
    MoveL Offs(pOrigin,108.8,29.4,0.0),vApproach,fine,tPen\WObj:=wPaper;
    MoveL Offs(pOrigin,108.6,29.2,0.0),vDraw,z1,tPen\WObj:=wPaper;
    MoveL Offs(pOrigin,108.4,29.2,0.0),vDraw,z1,tPen\WObj:=wPaper;
    MoveL Offs(pOrigin,108.2,29.4,0.0),vDraw,z1,tPen\WObj:=wPaper;
    MoveL Offs(pOrigin,108.2,29.6,0.0),vDraw,z1,tPen\WObj:=wPaper;
    MoveL Offs(pOrigin,108.4,29.7,0.0),vDraw,z1,tPen\WObj:=wPaper;
    MoveL Offs(pOrigin,108.4,30.1,0.0),vDraw,z1,tPen\WObj:=wPaper;
    MoveL Offs(pOrigin,108.6,30.3,0.0),vDraw,z1,tPen\WObj:=wPaper;
    MoveL Offs(pOrigin,108.8,30.1,0.0),vDraw,z1,tPen\WObj:=wPaper;
    MoveL Offs(pOrigin,108.8,29.4,0.0),vDraw,fine,tPen\WObj:=wPaper;
    MoveL Offs(pOrigin,108.8,29.4,15.0),vApproach,z5,tPen\WObj:=wPaper;
    MoveL Offs(pOrigin,107.8,29.9,15.0),vTravel,z5,tPen\WObj:=wPaper;
    MoveL Offs(pOrigin,107.8,29.9,0.0),vApproach,fine,tPen\WObj:=wPaper;
    MoveL Offs(pOrigin,107.1,29.4,0.0),vDraw,z1,tPen\WObj:=wPaper;
    MoveL Offs(pOrigin,106.9,29.4,0.0),vDraw,z1,tPen\WObj:=wPaper;
    MoveL Offs(pOrigin,106.7,29.6,0.0),vDraw,z1,tPen\WObj:=wPaper;
    MoveL Offs(pOrigin,106.7,29.9,0.0),vDraw,z1,tPen\WObj:=wPaper;
    MoveL Offs(pOrigin,106.5,30.1,0.0),vDraw,z1,tPen\WObj:=wPaper;
  ENDPROC

